# B&R Automation Studio project NAELD004C00R10L518F00 (part 7)

#### Act_OptP0001Startup.st
```iecst
ACTION Act_OptP0001Startup:

	//Screen Saver
	p_tyP0000SSaver ACCESS ADR(tyP0000SSaver.tySSaver);

	IF (eChgPage = UIP0001Startup) AND (eCurrPage = UIP0001Startup) THEN

		eStartupAct		:= StartupActRun;

		IF p_eStartupStat = StartupActRun AND p_eStartupStatus = Done THEN
			eStartupAct	:= StartupActIdle;

			IF p_bAlarmErr OR p_bAlarmWarning THEN
				eChgPage	:= UIP0600Alm;
			ELSE
				eChgPage	:= UIP0002Menu;
			END_IF

		END_IF

	END_IF

	tyP0001Startup.tyStartup.tyBarGraphStartup.iValue	:= DINT_TO_INT(p_eStartupStep + 1);
	tyP0001Startup.tyStartup.tyTxtStartupStat.sTxt		:= p_sStartupStepTxt;

	//IP Config
	IF DiagCpuIsSimulated() = FALSE THEN
		IF p_eStartupStep>1 THEN

			IF p_bStartupGetConfigDone THEN
				IF bTempAddrFillDone=FALSE THEN

					tyMcParamWr:= p_tyMcParamCurr;

					sTempIPAddr 	:= p_sHWInfoIPAddr;
					sTempSubnetMask	:= p_sHWInfoSubnetMask;
					udiTempEthMode	:= p_udiHWInfoEthMode;

					bTempAddrFillDone	:= TRUE;
				END_IF
			END_IF

			IF bTempAddrFillDone THEN

				IF bIPConfigChgDone=FALSE THEN

					IF  (p_tyMcParamCurr.eNetworkMod = UDINT_TO_DINT(udiTempEthMode)) AND (p_tyMcParamCurr.sIPAddr = sTempIPAddr) AND (p_tyMcParamCurr.sSubnetMask = sTempSubnetMask) THEN

						p_tyC0008MsgBox ACCESS ADR(tyP0001Startup.tyMsgBoxHide);
					ELSE
						IF p_bStartupMismatchSetConfigDone THEN

							IF (p_tyMcParamCurr.eNetworkMod <> UDINT_TO_DINT(udiTempEthMode)) THEN
								tyP0001Startup.tyMsgBoxIPConfig.tyTxtMsg.usiValueIdx := 114;
							ELSIF (p_tyMcParamCurr.sIPAddr <> sTempIPAddr) AND (p_tyMcParamCurr.sSubnetMask <> sTempSubnetMask) THEN
								tyP0001Startup.tyMsgBoxIPConfig.tyTxtMsg.usiValueIdx := 113;
							ELSIF (p_tyMcParamCurr.sIPAddr <> sTempIPAddr) THEN
								tyP0001Startup.tyMsgBoxIPConfig.tyTxtMsg.usiValueIdx := 111;
							ELSE
								tyP0001Startup.tyMsgBoxIPConfig.tyTxtMsg.usiValueIdx := 112;
							END_IF

							p_tyC0008MsgBox ACCESS ADR(tyP0001Startup.tyMsgBoxIPConfig);

						ELSE
							sSetIPAddr				:= p_tyMcParamCurr.sIPAddr;
							sSetSubnetMask			:= p_tyMcParamCurr.sSubnetMask;
							usiNetworkModeSelected	:= DINT_TO_USINT(p_tyMcParamCurr.eNetworkMod);

							bMismatchOverWriteConfig			:= TRUE;
						END_IF

					END_IF
				END_IF
			END_IF
		END_IF
	END_IF

	IF tyP0001Startup.tyMsgBoxIPConfig.tyBtnYes.bRtCompl = TRUE THEN
		tyP0001Startup.tyMsgBoxIPConfig.tyBtnYes.bRtCompl	:= FALSE;
		tyP0001Startup.tyMsgBoxIPConfig.tyBtnYes.bValue	:= FALSE;

		bIPConfigChgDone	:= TRUE;

		p_tyC0008MsgBox ACCESS ADR(tyP0001Startup.tyMsgBoxHide);

	ELSIF tyP0001Startup.tyMsgBoxIPConfig.tyBtnNo.bRtCompl = TRUE THEN

		IF (p_tyMcParamCurr.eNetworkMod <> UDINT_TO_DINT(udiTempEthMode))  THEN

			IF udiTempEthMode = DINT_TO_UDINT(IPFromDHCPServer) THEN

				bOverwriteEthMode	:= TRUE;
				bOverwriteIP 		:= FALSE;
				bOverwriteSubnet	:= FALSE;

				usiNetworkModeSelected	:= UDINT_TO_USINT(udiTempEthMode);

				tyMcParamWr.eNetworkMod	:= UDINT_TO_DINT(udiTempEthMode);

				bIPConfigChgDone	:= TRUE;

				tyP0001Startup.tyMsgBoxIPConfig.tyBtnNo.bRtCompl:= FALSE;
				tyP0001Startup.tyMsgBoxIPConfig.tyBtnNo.bValue	:= FALSE;

				p_tyC0008MsgBox ACCESS ADR(tyP0001Startup.tyMsgBoxHide);
			ELSE
				bOverwriteEthMode	:= TRUE;
				bOverwriteIP 		:= TRUE;
				bOverwriteSubnet	:= TRUE;

				usiNetworkModeSelected	:= UDINT_TO_USINT(udiTempEthMode);
				sSetIPAddr				:= sTempIPAddr;
				sSetSubnetMask			:= sTempSubnetMask;

				tyMcParamWr.eNetworkMod			:= UDINT_TO_DINT(udiTempEthMode);
				tyMcParamWr.sIPAddr				:= sTempIPAddr;
				tyMcParamWr.sSubnetMask			:= sTempSubnetMask;

				bIPConfigChgDone	:= TRUE;

				tyP0001Startup.tyMsgBoxIPConfig.tyBtnNo.bRtCompl:= FALSE;
				tyP0001Startup.tyMsgBoxIPConfig.tyBtnNo.bValue	:= FALSE;

				p_tyC0008MsgBox ACCESS ADR(tyP0001Startup.tyMsgBoxHide);
			END_IF

		ELSE

			IF (p_tyMcParamCurr.sIPAddr <> sTempIPAddr) AND (p_tyMcParamCurr.sSubnetMask <> sTempSubnetMask) THEN

				bOverwriteEthMode	:= FALSE;
				bOverwriteIP 		:= TRUE;
				bOverwriteSubnet	:= TRUE;

				sSetIPAddr		:= sTempIPAddr;
				sSetSubnetMask	:= sTempSubnetMask;

				tyMcParamWr.sIPAddr				:= sTempIPAddr;
				tyMcParamWr.sSubnetMask			:= sTempSubnetMask;

				bIPConfigChgDone	:= TRUE;

				tyP0001Startup.tyMsgBoxIPConfig.tyBtnNo.bRtCompl	:= FALSE;
				tyP0001Startup.tyMsgBoxIPConfig.tyBtnNo.bValue	:= FALSE;

				p_tyC0008MsgBox ACCESS ADR(tyP0001Startup.tyMsgBoxHide);

			ELSIF (p_tyMcParamCurr.sIPAddr <> sTempIPAddr) THEN

				bOverwriteEthMode	:= FALSE;
				bOverwriteIP 		:= TRUE;
				bOverwriteSubnet	:= FALSE;

				sSetIPAddr			:= sTempIPAddr;

				tyMcParamWr.sIPAddr	:= sTempIPAddr;

				bIPConfigChgDone	:= TRUE;

				tyP0001Startup.tyMsgBoxIPConfig.tyBtnNo.bRtCompl	:= FALSE;
				tyP0001Startup.tyMsgBoxIPConfig.tyBtnNo.bValue	:= FALSE;

				p_tyC0008MsgBox ACCESS ADR(tyP0001Startup.tyMsgBoxHide);
			ELSE

				bOverwriteEthMode	:= FALSE;
				bOverwriteIP 		:= FALSE;
				bOverwriteSubnet	:= TRUE;

				sSetSubnetMask	:= sTempSubnetMask;

				tyMcParamWr.sSubnetMask			:= sTempSubnetMask;

				bIPConfigChgDone				:= TRUE;

				tyP0001Startup.tyMsgBoxIPConfig.tyBtnNo.bRtCompl	:= FALSE;
				tyP0001Startup.tyMsgBoxIPConfig.tyBtnNo.bValue		:= FALSE;

				p_tyC0008MsgBox ACCESS ADR(tyP0001Startup.tyMsgBoxHide);
			END_IF
		END_IF
	END_IF

	//new for Hermes 1.3
	IF p_eStartupStep = StartupStepHermes AND p_bWaitDecision AND p_tyNtParamCurr.bHermesSvyPrep AND p_tyMcParamCurr.bHermesSvyEn AND p_tyNtParamCurr.bHermesSvyFirstMcInTheLine AND p_tyHermesConfiguration.tySvyParam.bFeatureQueryWorkOrderInfo THEN
		p_tyC0008MsgBox ACCESS ADR(tyP0001Startup.tyMsgBoxWorkOrder);

		IF tyP0001Startup.tyMsgBoxWorkOrder.tyBtnYes.bRtCompl = TRUE THEN
			tyP0001Startup.tyMsgBoxWorkOrder.tyBtnYes.bRtCompl	:= FALSE;
			bReadWorkOrder :=TRUE;
		END_IF

		IF tyP0001Startup.tyMsgBoxWorkOrder.tyBtnNo.bRtCompl = TRUE THEN
			tyP0001Startup.tyMsgBoxWorkOrder.tyBtnNo.bRtCompl	:= FALSE;
			bSkipWorkOrder :=TRUE;
		END_IF

		IF bReadWorkOrder OR bSkipWorkOrder THEN
			p_tyC0008MsgBox ACCESS ADR(tyP0001Startup.tyMsgBoxHide);
		END_IF

	ELSIF p_eStartupStep = StartupStepHermes AND p_bWaitDecision AND (p_tyNtParamCurr.bHermesSvyPrep = FALSE OR p_tyMcParamCurr.bHermesSvyEn = FALSE OR p_tyNtParamCurr.bHermesSvyFirstMcInTheLine = FALSE OR p_tyHermesConfiguration.tySvyParam.bFeatureQueryWorkOrderInfo = FALSE) THEN
		p_tyC0008MsgBox ACCESS ADR(tyP0001Startup.tyMsgBoxHide);
		bReadWorkOrder :=FALSE;
		bSkipWorkOrder :=TRUE;
	END_IF

END_ACTION
```

#### Act_EntP0002Disp.st
```iecst
ACTION Act_EntP0002Disp:

	//Access
	p_tyC0005Main ACCESS ADR(tyCommon.tyMain);

	p_tyC0007Notif ACCESS ADR(tyCommon.tyNotif);

	IF NOT bPromptSessionExp THEN
		p_tyC0008MsgBox ACCESS ADR(tyP0002Menu.tyMsgBoxHide);
	END_IF

	p_tyC0009Info ACCESS ADR(tyCommon.tyInfo);

	p_tyP0002Menu ACCESS ADR(tyP0002Menu.tyMenu);

	//Display
	//Leader Follower
	IF p_tyNtParamCurr.bLFPrep = TRUE AND p_tyMcParamCurr.bLFEn = TRUE AND ((NOT p_tyNtParamCurr.bLFUsrSetPrep AND p_tyNtParamCurr.bLeaderMc) OR (p_tyNtParamCurr.bLFUsrSetPrep AND p_tyMcParamCurr.bLFLeaderMc)) THEN
		fUIInRtStatOff(ADR(tyP0002Menu.tyMenu.tyBtnLFSet.uiRtStat));
		fUIInRtStatOff(ADR(tyP0002Menu.tyMenu.tyBtnLFCtrl.uiRtStat));
	ELSE
		fUIInRtStatHide(ADR(tyP0002Menu.tyMenu.tyBtnLFSet.uiRtStat));
		fUIInRtStatHide(ADR(tyP0002Menu.tyMenu.tyBtnLFCtrl.uiRtStat));
	END_IF

//	tyP0002Menu.tyMenu.tyBtnSimu.uiRtStat.0 := NOT(p_tyNtParamCurr.bProjAGVPrep AND p_tyMcParamCurr.bAGVComEn);

	//Login Logout Display
	IF bLoginSuccess = FALSE THEN
		tyP0002Menu.tyMenu.tyBtnLogin.usiBitmapIdx	:= 0;
		tyP0002Menu.tyMenu.tyBtnLogin.usiTxtIdx		:= 0;
	ELSE
		tyP0002Menu.tyMenu.tyBtnLogin.usiBitmapIdx	:= 1;
		tyP0002Menu.tyMenu.tyBtnLogin.usiTxtIdx		:= 1;
	END_IF

	//Mask
	Act_OptP0002Mask;
	bTeachServo := FALSE;
END_ACTION
```

#### Act_OptP0002ChgPage.st
```iecst
ACTION Act_OptP0002ChgPage:

	//General
	IF tyP0002Menu.tyMenu.tyBtnOpt.bRtCompl = TRUE THEN
		tyP0002Menu.tyMenu.tyBtnOpt.bRtCompl				:= FALSE;
		eChgPage											:= UIP0200OpsGen;

	ELSIF tyP0002Menu.tyMenu.tyBtnProdSel.bRtCompl = TRUE THEN
		tyP0002Menu.tyMenu.tyBtnProdSel.bRtCompl			:= FALSE;
		eChgPage											:= UIP0400ProdSel;

	ELSIF tyP0002Menu.tyMenu.tyBtnMagSel.bRtCompl = TRUE THEN
		tyP0002Menu.tyMenu.tyBtnMagSel.bRtCompl				:= FALSE;
		eChgPage											:= UIP0410MagSel;

	ELSIF tyP0002Menu.tyMenu.tyBtnMcInfo.bRtCompl = TRUE THEN
		tyP0002Menu.tyMenu.tyBtnMcInfo.bRtCompl				:= FALSE;
		eChgPage											:= UIP0300McInfo;

	ELSIF tyP0002Menu.tyMenu.tyBtnAlm.bRtCompl = TRUE THEN
		tyP0002Menu.tyMenu.tyBtnAlm.bRtCompl				:= FALSE;
		eChgPage											:= UIP0600Alm;

	ELSIF tyP0002Menu.tyMenu.tyBtnLogin.bRtCompl = TRUE THEN
		tyP0002Menu.tyMenu.tyBtnLogin.bRtCompl				:= FALSE;
		eChgPage											:= UIP0100Login;

	ELSIF tyP0002Menu.tyMenu.tyBtnLFCtrl.bRtCompl = TRUE THEN
		tyP0002Menu.tyMenu.tyBtnLFCtrl.bRtCompl				:= FALSE;
		eChgPage											:= UIP0700LFCtrl;

	ELSIF tyP0002Menu.tyMenu.tyBtnMagInfo.bRtCompl = TRUE THEN
		tyP0002Menu.tyMenu.tyBtnMagInfo.bRtCompl			:= FALSE;
		eChgPage											:= UIP0800MagInfo;

	//Manual
	ELSIF tyP0002Menu.tyMenu.tyBtnGenInput.bRtCompl = TRUE THEN
		bUIManualMod										:= TRUE;
		tyP0002Menu.tyMenu.tyBtnGenInput.bRtCompl			:= FALSE;
		eChgPage											:= UIP0900GenIn;

	ELSIF tyP0002Menu.tyMenu.tyBtnGenOutput.bRtCompl = TRUE THEN
		bUIManualMod										:= TRUE;
		tyP0002Menu.tyMenu.tyBtnGenOutput.bRtCompl			:= FALSE;
		eChgPage											:= UIP0910GenOut;

	ELSIF tyP0002Menu.tyMenu.tyBtnMovCtrl.bRtCompl = TRUE THEN
		bUIManualMod										:= TRUE;
		tyP0002Menu.tyMenu.tyBtnMovCtrl.bRtCompl			:= FALSE;
		eChgPage											:= UIP0920MtrNPneuCtrl;

	ELSIF tyP0002Menu.tyMenu.tyBtnCommCtrl.bRtCompl = TRUE THEN
		bUIManualMod										:= TRUE;
		tyP0002Menu.tyMenu.tyBtnCommCtrl.bRtCompl			:= FALSE;
		eChgPage											:= UIP0940CommCtrl;

	ELSIF tyP0002Menu.tyMenu.tyBtnSimu.bRtCompl = TRUE THEN
		tyP0002Menu.tyMenu.tyBtnSimu.bRtCompl				:= FALSE;
		eChgPage											:= UIP0950Simu;

	//Settings
	ELSIF tyP0002Menu.tyMenu.tyBtnLang.bRtCompl = TRUE THEN
		tyP0002Menu.tyMenu.tyBtnLang.bRtCompl				:= FALSE;
		eChgPage											:= UIP1000Lang;

	ELSIF tyP0002Menu.tyMenu.tyBtnMcSet.bRtCompl = TRUE THEN
		tyP0002Menu.tyMenu.tyBtnMcSet.bRtCompl				:= FALSE;
		eChgPage											:= UIP1020McSetNavi;

	ELSIF tyP0002Menu.tyMenu.tyBtnMagSet.bRtCompl = TRUE THEN
		tyP0002Menu.tyMenu.tyBtnMagSet.bRtCompl				:= FALSE;
		eChgPage											:= UIP1030MagSet;

	ELSIF tyP0002Menu.tyMenu.tyBtnProdSet.bRtCompl = TRUE THEN
		tyP0002Menu.tyMenu.tyBtnProdSet.bRtCompl			:= FALSE;
		eChgPage											:= UIP1040ProdSet;

	ELSIF tyP0002Menu.tyMenu.tyBtnLFSet.bRtCompl = TRUE THEN
		tyP0002Menu.tyMenu.tyBtnLFSet.bRtCompl				:= FALSE;
		eChgPage											:= UIP1050LFSet;

	ELSIF tyP0002Menu.tyMenu.tyBtnUsrMgmt.bRtCompl = TRUE THEN
		tyP0002Menu.tyMenu.tyBtnUsrMgmt.bRtCompl			:= FALSE;
		eChgPage											:= UIP1080UsrMgmt;

	END_IF
	fbActSimuTmr (IN:= tyP0002Menu.tyMenu.tyBtnHotspotActSimu.bValue = TRUE ,PT:=T#8s);
	IF fbActSimuTmr.Q THEN
		IF tyP0002Menu.tyMenu.tyBtnSimu.uiRtStat =0 THEN
			tyP0002Menu.tyMenu.tyBtnSimu.uiRtStat := 1;
			fbActSimuTmr (IN:= FALSE);
		ELSE
			tyP0002Menu.tyMenu.tyBtnSimu.uiRtStat := 0;
			fbActSimuTmr (IN:= FALSE);
		END_IF
	END_IF

END_ACTION
```

#### Act_OptP0002Mask.st
```iecst
ACTION Act_OptP0002Mask:

	tyP0002Menu.tyMenu.tyBtnOpt.uiMaskRtStat.0 					:= p_tyUsrMgmtCurrAccessRgt.bOpt;
	tyP0002Menu.tyMenu.tyBtnMcInfo.uiMaskRtStat.0 				:= p_tyUsrMgmtCurrAccessRgt.bMcInfo;
	tyP0002Menu.tyMenu.tyBtnMagInfo.uiMaskRtStat.0				:= p_tyUsrMgmtCurrAccessRgt.bMagInfo;
	tyP0002Menu.tyMenu.tyBtnAlm.uiMaskRtStat.0 					:= p_tyUsrMgmtCurrAccessRgt.bAlm;
	tyP0002Menu.tyMenu.tyBtnLogin.uiMaskRtStat.0				:= p_bOpsStatusStop;
	tyP0002Menu.tyMenu.tyBtnLFCtrl.uiMaskRtStat.0 				:= p_tyUsrMgmtCurrAccessRgt.bLFCtrl;
	tyP0002Menu.tyMenu.tyBtnGenInput.uiMaskRtStat.0				:= p_tyUsrMgmtCurrAccessRgt.bManual AND p_bOpsStatusStop;
	tyP0002Menu.tyMenu.tyBtnGenOutput.uiMaskRtStat.0			:= p_tyUsrMgmtCurrAccessRgt.bManual AND p_bOpsStatusStop;
	tyP0002Menu.tyMenu.tyBtnMovCtrl.uiMaskRtStat.0 				:= p_tyUsrMgmtCurrAccessRgt.bManual AND p_bOpsStatusStop;
	tyP0002Menu.tyMenu.tyBtnCommCtrl.uiMaskRtStat.0 			:= p_tyUsrMgmtCurrAccessRgt.bManual AND p_bOpsStatusStop;
	tyP0002Menu.tyMenu.tyBtnSimu.uiMaskRtStat.0 				:= p_tyUsrMgmtCurrAccessRgt.bSimulation AND p_bOpsStatusStop;
	tyP0002Menu.tyMenu.tyBtnProdSet.uiMaskRtStat.0 				:= p_tyUsrMgmtCurrAccessRgt.bProdSet AND p_bOpsStatusStop;
	tyP0002Menu.tyMenu.tyBtnMagSet.uiMaskRtStat.0				:= p_tyUsrMgmtCurrAccessRgt.bMagSet AND p_bOpsStatusStop;
	tyP0002Menu.tyMenu.tyBtnMcSet.uiMaskRtStat.0 				:= p_tyUsrMgmtCurrAccessRgt.bMcSet AND p_bOpsStatusStop;
	tyP0002Menu.tyMenu.tyBtnLang.uiMaskRtStat.0 				:= p_tyUsrMgmtCurrAccessRgt.bLang AND p_bOpsStatusStop;
	tyP0002Menu.tyMenu.tyBtnUsrMgmt.uiMaskRtStat.0 				:= p_tyUsrMgmtCurrAccessRgt.bUsrMgmt AND p_bOpsStatusStop;
	tyP0002Menu.tyMenu.tyBtnLFSet.uiMaskRtStat.0 				:= p_tyUsrMgmtCurrAccessRgt.bLFSet AND p_bOpsStatusStop;

	tyP0002Menu.tyMenu.tyBitmapMaskProdSetLCS.uiMaskRtStat.0	:= NOT(p_tyNtParamCurr.bLCSManageRcpPrep AND p_tyMcParamCurr.bLCSManageRcpEn);

//	IF p_tyNtParamCurr.eProjMag = LDMagTriple THEN
//		tyP0002Menu.tyMenu.tyBtnProdSel.uiMaskRtStat.0 	:= p_tyUsrMgmtCurrAccessRgt.bProdSel AND p_bOpsStatusStop AND NOT(p_bBuffer1MagPresent OR p_bBuffer2MagPresent OR p_bBuffer3MagPresent);
//		tyP0002Menu.tyMenu.tyBtnMagSel.uiMaskRtStat.0	:= p_tyUsrMgmtCurrAccessRgt.bMagSel AND p_bOpsStatusStop AND NOT(p_bBuffer1MagPresent OR p_bBuffer2MagPresent OR p_bBuffer3MagPresent);
//	ELSE
//		tyP0002Menu.tyMenu.tyBtnProdSel.uiMaskRtStat.0 	:= p_tyUsrMgmtCurrAccessRgt.bProdSel AND p_bOpsStatusStop AND NOT(p_bBuffer1MagPresent OR p_bBuffer2MagPresent);
//		tyP0002Menu.tyMenu.tyBtnMagSel.uiMaskRtStat.0	:= p_tyUsrMgmtCurrAccessRgt.bMagSel AND p_bOpsStatusStop AND NOT(p_bBuffer1MagPresent OR p_bBuffer2MagPresent);
//	END_IF

	IF p_tyNtParamCurr.eProjMag = LDMagTriple THEN
		tyP0002Menu.tyMenu.tyBtnProdSel.uiMaskRtStat.0 	:= p_bOpsStatusStop AND NOT(p_bBuffer1MagPresent OR p_bBuffer2MagPresent OR p_bBuffer3MagPresent);
		tyP0002Menu.tyMenu.tyBtnMagSel.uiMaskRtStat.0	:= p_bOpsStatusStop AND NOT(p_bBuffer1MagPresent OR p_bBuffer2MagPresent OR p_bBuffer3MagPresent);
	ELSIF p_tyNtParamCurr.eProjMag = LDMagQuadruple THEN
		tyP0002Menu.tyMenu.tyBtnProdSel.uiMaskRtStat.0 	:= p_bOpsStatusStop AND NOT(p_bBuffer1MagPresent OR p_bBuffer2MagPresent OR p_bBuffer3MagPresent OR p_bBuffer4MagPresent);
		tyP0002Menu.tyMenu.tyBtnMagSel.uiMaskRtStat.0	:= p_bOpsStatusStop AND NOT(p_bBuffer1MagPresent OR p_bBuffer2MagPresent OR p_bBuffer3MagPresent OR p_bBuffer4MagPresent);

	ELSE
		tyP0002Menu.tyMenu.tyBtnProdSel.uiMaskRtStat.0 	:= p_bOpsStatusStop AND NOT(p_bBuffer1MagPresent OR p_bBuffer2MagPresent);
		tyP0002Menu.tyMenu.tyBtnMagSel.uiMaskRtStat.0	:= p_bOpsStatusStop AND NOT(p_bBuffer1MagPresent OR p_bBuffer2MagPresent);
	END_IF
END_ACTION
```

#### Act_OptP0002MsgGuide.st
```iecst
ACTION Act_OptP0002MsgGuide:

	//Display
	tyP0002Menu.tyMenu.tyHotspotProdSel.uiRtStat.0	:= tyP0002Menu.tyMenu.tyBtnProdSel.uiMaskRtStat.0;
	tyP0002Menu.tyMenu.tyHotspotMagSel.uiRtStat.0	:= tyP0002Menu.tyMenu.tyBtnMagSel.uiMaskRtStat.0;

	IF p_tyNtParamCurr.eProjMag = LDMagTriple THEN
		tyP0002Menu.tyMenu.tyHotspotProdSel.bRtLk	:= NOT(p_bBuffer1MagPresent OR p_bBuffer2MagPresent OR p_bBuffer3MagPresent);
		tyP0002Menu.tyMenu.tyHotspotMagSel.bRtLk	:= NOT(p_bBuffer1MagPresent OR p_bBuffer2MagPresent OR p_bBuffer3MagPresent);
	ELSE
		tyP0002Menu.tyMenu.tyHotspotProdSel.bRtLk	:= NOT(p_bBuffer1MagPresent OR p_bBuffer2MagPresent);
		tyP0002Menu.tyMenu.tyHotspotMagSel.bRtLk	:= NOT(p_bBuffer1MagPresent OR p_bBuffer2MagPresent);
	END_IF

	//Control
	IF tyP0002Menu.tyMenu.tyHotspotProdSel.bRtCompl OR tyP0002Menu.tyMenu.tyHotspotMagSel.bRtCompl THEN
		p_tyC0008MsgBox ACCESS ADR(tyP0002Menu.tyMsgBoxRemoveMag);

		IF tyP0002Menu.tyMsgBoxRemoveMag.tyBtnNo.bRtCompl = TRUE THEN
			tyP0002Menu.tyMsgBoxRemoveMag.tyBtnNo.bRtCompl	:= FALSE;
			tyP0002Menu.tyMsgBoxRemoveMag.tyBtnNo.bValue	:= FALSE;

			p_tyC0008MsgBox ACCESS ADR(tyP0002Menu.tyMsgBoxHide);

			IF tyP0002Menu.tyMenu.tyHotspotProdSel.bRtCompl AND tyP0002Menu.tyMenu.tyBtnProdSel.uiMaskRtStat.0 THEN
				eChgPage	:= UIP0400ProdSel;

			ELSIF tyP0002Menu.tyMenu.tyHotspotMagSel.bRtCompl AND tyP0002Menu.tyMenu.tyBtnMagSel.uiMaskRtStat.0 THEN
				eChgPage	:= UIP0410MagSel;

			END_IF

			tyP0002Menu.tyMenu.tyHotspotProdSel.bRtCompl	:= FALSE;
			tyP0002Menu.tyMenu.tyHotspotMagSel.bRtCompl		:= FALSE;

		END_IF

	END_IF

END_ACTION
```

#### Act_OptP0002ToP1081UnlockCoverPB.st
```iecst
ACTION Act_OptP0002ToP1081UnlockCoverPB:

	IF p_tyDI.bDSUnlockCoverSig AND (p_bOpsTravLifStandby OR p_bOpsRun = FALSE) AND p_ePullConvStatus <> Busy THEN
		bMachineSafetySigToDS := TRUE;																						//
	ELSE
		bMachineSafetySigToDS := FALSE;																						//
	END_IF

END_ACTION
```

#### Act_EntP0200Disp.st
```iecst
ACTION Act_EntP0200Disp:

	//Access Address
	p_tyC0005Main ACCESS ADR(tyCommon.tyMain);

	p_tyC0007Notif ACCESS ADR(tyCommon.tyNotif);

	p_tyC0008MsgBox ACCESS ADR(tyP0200OpsGen.tyMsgBoxHide);

	p_tyC0009Info ACCESS ADR(tyCommon.tyInfo);

	p_tyC0010RcyMsg ACCESS ADR(tyP0200OpsGen.tyRcyMsgHide);

	p_tyP0200OpsGen ACCESS ADR(tyP0200OpsGen.tyOps);
	p_tyP0200OpsDSCommB ACCESS ADR(tyP0200OpsGen.tyDSCommB);

	p_tyP0200OpsDSAVSMEMA ACCESS ADR(tyP0200OpsGen.tyDSAVSMEMA);
	p_tyP0200OpsDSBVSMEMA ACCESS ADR(tyP0200OpsGen.tyDSBVSMEMA);
	p_tyP0200OpsDSAVSMEMA1 ACCESS ADR(tyP0200OpsGen.tyDSAVSMEMA1);
	p_tyP0200OpsDSBVSMEMA1 ACCESS ADR(tyP0200OpsGen.tyDSBVSMEMA1);
	p_tyP0200OpsBypsInitConv ACCESS ADR(tyP0200OpsGen.tyBypsInitConv);

	p_tyP0200OpsBarCodeScan ACCESS ADR(tyP0200OpsGen.tyBarCodeScan);
	//Display
	//Downstream A
	IF p_tyMcParamCurr.eDSCommA = McSetCommModHermes THEN
		tyP0200OpsGen.tyOps.tyBitmapDSAComm.usiValueIdx	:= 1;
		tyP0200OpsGen.tyOps.tyBitmapDSAComm1.usiValueIdx	:= 1;
	ELSIF p_tyMcParamCurr.eDSCommA = McSetCommModSMEMA THEN
		tyP0200OpsGen.tyOps.tyBitmapDSAComm.usiValueIdx	:= 0;
		tyP0200OpsGen.tyOps.tyBitmapDSAComm1.usiValueIdx	:= 0;
	END_IF

	//Downstream B
	IF p_tyMcParamCurr.eDSCommB = McSetCommModHermes THEN
		tyP0200OpsGen.tyDSCommB.tyBitmapDSBComm.usiValueIdx	:= 1;
		tyP0200OpsGen.tyDSCommB.tyBitmapDSBComm1.usiValueIdx	:= 1;
	ELSIF p_tyMcParamCurr.eDSCommB = McSetCommModSMEMA THEN
		tyP0200OpsGen.tyDSCommB.tyBitmapDSBComm.usiValueIdx	:= 0;
		tyP0200OpsGen.tyDSCommB.tyBitmapDSBComm1.usiValueIdx	:= 0;
	END_IF

	//Virtual SMEMA
	IF (p_tyUsrMgmtCurrUsr.eUsrLvl = UsrMgmtLvl1) OR p_tyNtParamCurr.bVSMEMAPrep = FALSE OR p_tyMcParamCurr.bVSMEMAEn = FALSE OR (p_tyMcParamCurr.eDSCommA = McSetCommModHermes AND p_tyMcParamCurr.eDSCommB = McSetCommModHermes) THEN

		tyP0200OpsGen.tyOps.tyHotspotDSAVSMEMA.bValue		:= FALSE;
		tyP0200OpsGen.tyDSCommB.tyHotspotDSBVSMEMA.bValue	:= FALSE;
		tyP0200OpsGen.tyOps.tyHotspotDSAVSMEMA1.bValue		:= FALSE;
		tyP0200OpsGen.tyDSCommB.tyHotspotDSBVSMEMA1.bValue	:= FALSE;

		memset(ADR(tyP0200OpsGen.tyDSAVSMEMA), 0, SIZEOF(tyP0200OpsGen.tyDSAVSMEMA));
		memset(ADR(tyP0200OpsGen.tyDSBVSMEMA), 0, SIZEOF(tyP0200OpsGen.tyDSBVSMEMA));
		memset(ADR(tyP0200OpsGen.tyDSAVSMEMA1), 0, SIZEOF(tyP0200OpsGen.tyDSAVSMEMA1));
		memset(ADR(tyP0200OpsGen.tyDSBVSMEMA1), 0, SIZEOF(tyP0200OpsGen.tyDSBVSMEMA1));

		fUIInRtStatHide(ADR(tyP0200OpsGen.tyOps.tyHotspotDSAVSMEMA.uiRtStat));
		fUIInRtStatHide(ADR(tyP0200OpsGen.tyDSCommB.tyHotspotDSBVSMEMA.uiRtStat));
		fUIInRtStatHide(ADR(tyP0200OpsGen.tyDSAVSMEMA.tyLyr.uiRtStat));
		fUIInRtStatHide(ADR(tyP0200OpsGen.tyDSBVSMEMA.tyLyr.uiRtStat));

		fUIInRtStatHide(ADR(tyP0200OpsGen.tyOps.tyHotspotDSAVSMEMA1.uiRtStat));
		fUIInRtStatHide(ADR(tyP0200OpsGen.tyDSCommB.tyHotspotDSBVSMEMA1.uiRtStat));
		fUIInRtStatHide(ADR(tyP0200OpsGen.tyDSAVSMEMA1.tyLyr.uiRtStat));
		fUIInRtStatHide(ADR(tyP0200OpsGen.tyDSBVSMEMA1.tyLyr.uiRtStat));

		bVSMEMADSAEn	:= FALSE;
		bVSMEMADSBEn	:= FALSE;
	ELSE

		//Downstream A
		IF p_tyMcParamCurr.eDSCommA = McSetCommModHermes THEN
			tyP0200OpsGen.tyOps.tyHotspotDSAVSMEMA.bValue	:= FALSE;
			tyP0200OpsGen.tyOps.tyHotspotDSAVSMEMA1.bValue	:= FALSE;

			memset(ADR(tyP0200OpsGen.tyDSAVSMEMA), 0, SIZEOF(tyP0200OpsGen.tyDSAVSMEMA));

			fUIInRtStatHide(ADR(tyP0200OpsGen.tyOps.tyHotspotDSAVSMEMA.uiRtStat));
			fUIInRtStatHide(ADR(tyP0200OpsGen.tyDSAVSMEMA.tyLyr.uiRtStat));

			memset(ADR(tyP0200OpsGen.tyDSAVSMEMA1), 0, SIZEOF(tyP0200OpsGen.tyDSAVSMEMA1));

			fUIInRtStatHide(ADR(tyP0200OpsGen.tyOps.tyHotspotDSAVSMEMA1.uiRtStat));
			fUIInRtStatHide(ADR(tyP0200OpsGen.tyDSAVSMEMA1.tyLyr.uiRtStat));

		ELSIF p_tyMcParamCurr.eDSCommA = McSetCommModSMEMA THEN
			IF p_tyNtParamCurr.bUIConvDirRL = FALSE THEN //LR
				fUIInRtStatOff(ADR(tyP0200OpsGen.tyOps.tyHotspotDSAVSMEMA.uiRtStat));

				fUIInRtStatHide(ADR(tyP0200OpsGen.tyOps.tyHotspotDSAVSMEMA1.uiRtStat));
				fUIInRtStatHide(ADR(tyP0200OpsGen.tyOps.tyTxtLane1.uiRtStat));
				fUIInRtStatHide(ADR(tyP0200OpsGen.tyOps.tyBitmapDSIn1.uiRtStat));
				fUIInRtStatHide(ADR(tyP0200OpsGen.tyOps.tyBitmapDSOut1.uiRtStat));
				fUIInRtStatHide(ADR(tyP0200OpsGen.tyOps.tyBitmapDSAComm1.uiRtStat));
				memset(ADR(tyP0200OpsGen.tyDSAVSMEMA1), 0, SIZEOF(tyP0200OpsGen.tyDSAVSMEMA1));
				fUIInRtStatHide(ADR(tyP0200OpsGen.tyDSAVSMEMA1.tyLyr.uiRtStat));
			ELSE //RL
				fUIInRtStatOff(ADR(tyP0200OpsGen.tyOps.tyHotspotDSAVSMEMA1.uiRtStat));

				fUIInRtStatHide(ADR(tyP0200OpsGen.tyOps.tyHotspotDSAVSMEMA.uiRtStat));
				fUIInRtStatHide(ADR(tyP0200OpsGen.tyOps.tyTxtLane.uiRtStat));
				fUIInRtStatHide(ADR(tyP0200OpsGen.tyOps.tyBitmapDSIn.uiRtStat));
				fUIInRtStatHide(ADR(tyP0200OpsGen.tyOps.tyBitmapDSOut.uiRtStat));
				fUIInRtStatHide(ADR(tyP0200OpsGen.tyOps.tyBitmapDSAComm.uiRtStat));
				memset(ADR(tyP0200OpsGen.tyDSAVSMEMA), 0, SIZEOF(tyP0200OpsGen.tyDSAVSMEMA));
				fUIInRtStatHide(ADR(tyP0200OpsGen.tyDSAVSMEMA.tyLyr.uiRtStat));

			END_IF

		END_IF

		//Downstream B
		IF p_tyNtParamCurr.bProjLaneBPrep THEN
			IF p_tyMcParamCurr.eDSCommB = McSetCommModHermes THEN
				tyP0200OpsGen.tyDSCommB.tyHotspotDSBVSMEMA.bValue	:= FALSE;
				tyP0200OpsGen.tyDSCommB.tyHotspotDSBVSMEMA1.bValue	:= FALSE;

				memset(ADR(tyP0200OpsGen.tyDSBVSMEMA), 0, SIZEOF(tyP0200OpsGen.tyDSBVSMEMA));
				fUIInRtStatHide(ADR(tyP0200OpsGen.tyDSCommB.tyHotspotDSBVSMEMA.uiRtStat));
				fUIInRtStatHide(ADR(tyP0200OpsGen.tyDSBVSMEMA.tyLyr.uiRtStat));

				memset(ADR(tyP0200OpsGen.tyDSBVSMEMA1), 0, SIZEOF(tyP0200OpsGen.tyDSBVSMEMA1));
				fUIInRtStatHide(ADR(tyP0200OpsGen.tyDSCommB.tyHotspotDSBVSMEMA1.uiRtStat));
				fUIInRtStatHide(ADR(tyP0200OpsGen.tyDSBVSMEMA1.tyLyr.uiRtStat));

			ELSIF p_tyMcParamCurr.eDSCommB = McSetCommModSMEMA THEN
				IF p_tyNtParamCurr.bUIConvDirRL = FALSE THEN //LR
					fUIInRtStatOff(ADR(tyP0200OpsGen.tyDSCommB.tyHotspotDSBVSMEMA.uiRtStat));

					fUIInRtStatHide(ADR(tyP0200OpsGen.tyDSCommB.tyHotspotDSBVSMEMA1.uiRtStat));
					fUIInRtStatHide(ADR(tyP0200OpsGen.tyDSCommB.tyTxtLane1.uiRtStat));
					fUIInRtStatHide(ADR(tyP0200OpsGen.tyDSCommB.tyBitmapIn1.uiRtStat));
					fUIInRtStatHide(ADR(tyP0200OpsGen.tyDSCommB.tyBitmapOut1.uiRtStat));
					fUIInRtStatHide(ADR(tyP0200OpsGen.tyDSCommB.tyBitmapDSBComm1.uiRtStat));
					fUIInRtStatHide(ADR(tyP0200OpsGen.tyDSBVSMEMA1.tyLyr.uiRtStat));

				ELSE
					fUIInRtStatOff(ADR(tyP0200OpsGen.tyDSCommB.tyHotspotDSBVSMEMA1.uiRtStat));

					fUIInRtStatHide(ADR(tyP0200OpsGen.tyDSCommB.tyHotspotDSBVSMEMA.uiRtStat));
					fUIInRtStatHide(ADR(tyP0200OpsGen.tyDSCommB.tyTxtLane.uiRtStat));
					fUIInRtStatHide(ADR(tyP0200OpsGen.tyDSCommB.tyBitmapIn.uiRtStat));
					fUIInRtStatHide(ADR(tyP0200OpsGen.tyDSCommB.tyBitmapOut.uiRtStat));
					fUIInRtStatHide(ADR(tyP0200OpsGen.tyDSCommB.tyBitmapDSBComm.uiRtStat));
					fUIInRtStatHide(ADR(tyP0200OpsGen.tyDSBVSMEMA.tyLyr.uiRtStat));
				END_IF

			END_IF

		END_IF

	END_IF

	//Conveyor Direction - SMEMA Arrow Indicator
	IF p_tyNtParamCurr.bUIConvDirRL THEN
		fUIInRtStatHide(ADR(tyP0200OpsGen.tyOps.tyBitmapDSIn.uiRtStat));
		fUIInRtStatHide(ADR(tyP0200OpsGen.tyOps.tyBitmapDSOut.uiRtStat));
		fUIInRtStatHide(ADR(tyP0200OpsGen.tyOps.tyTxtLane.uiRtStat));
		fUIInRtStatHide(ADR(tyP0200OpsGen.tyOps.tyHotspotDSAVSMEMA.uiRtStat));
		fUIInRtStatHide(ADR(tyP0200OpsGen.tyOps.tyBitmapDSAComm.uiRtStat));
		fUIInRtStatHide(ADR(tyP0200OpsGen.tyOps.tyBitmapDSAComm.uiMaskRtStat));

		fUIInRtStatHide(ADR(tyP0200OpsGen.tyDSCommB.tyBitmapIn.uiRtStat));
		fUIInRtStatHide(ADR(tyP0200OpsGen.tyDSCommB.tyBitmapOut.uiRtStat));
		fUIInRtStatHide(ADR(tyP0200OpsGen.tyDSCommB.tyTxtLane.uiRtStat));
		fUIInRtStatHide(ADR(tyP0200OpsGen.tyDSCommB.tyHotspotDSBVSMEMA.uiRtStat));
		fUIInRtStatHide(ADR(tyP0200OpsGen.tyDSCommB.tyBitmapDSBComm.uiRtStat));
		fUIInRtStatHide(ADR(tyP0200OpsGen.tyDSCommB.tyBitmapDSBComm.uiMaskRtStat));

		fUIInRtStatOff(ADR(tyP0200OpsGen.tyOps.tyBitmapDSIn1.uiRtStat));
		fUIInRtStatOff(ADR(tyP0200OpsGen.tyOps.tyBitmapDSOut1.uiRtStat));
		fUIInRtStatOff(ADR(tyP0200OpsGen.tyOps.tyTxtLane1.uiRtStat));
		fUIInRtStatOff(ADR(tyP0200OpsGen.tyOps.tyHotspotDSAVSMEMA1.uiRtStat));
		fUIInRtStatOff(ADR(tyP0200OpsGen.tyOps.tyBitmapDSAComm1.uiRtStat));
		fUIInRtStatOff(ADR(tyP0200OpsGen.tyOps.tyBitmapDSAComm1.uiMaskRtStat));

		fUIInRtStatOff(ADR(tyP0200OpsGen.tyDSCommB.tyBitmapIn1.uiRtStat));
		fUIInRtStatOff(ADR(tyP0200OpsGen.tyDSCommB.tyBitmapOut1.uiRtStat));
		fUIInRtStatOff(ADR(tyP0200OpsGen.tyDSCommB.tyTxtLane1.uiRtStat));
		fUIInRtStatOff(ADR(tyP0200OpsGen.tyDSCommB.tyHotspotDSBVSMEMA1.uiRtStat));
		fUIInRtStatOff(ADR(tyP0200OpsGen.tyDSCommB.tyBitmapDSBComm1.uiRtStat));
		fUIInRtStatOff(ADR(tyP0200OpsGen.tyDSCommB.tyBitmapDSBComm1.uiMaskRtStat));

	ELSE // LR

		fUIInRtStatOff(ADR(tyP0200OpsGen.tyOps.tyBitmapDSIn.uiRtStat));
		fUIInRtStatOff(ADR(tyP0200OpsGen.tyOps.tyBitmapDSOut.uiRtStat));
		fUIInRtStatOff(ADR(tyP0200OpsGen.tyOps.tyTxtLane.uiRtStat));
		fUIInRtStatOff(ADR(tyP0200OpsGen.tyOps.tyHotspotDSAVSMEMA.uiRtStat));
		fUIInRtStatOff(ADR(tyP0200OpsGen.tyOps.tyBitmapDSAComm.uiRtStat));
		fUIInRtStatOff(ADR(tyP0200OpsGen.tyOps.tyBitmapDSAComm.uiMaskRtStat));

		fUIInRtStatOff(ADR(tyP0200OpsGen.tyDSCommB.tyBitmapIn.uiRtStat));
		fUIInRtStatOff(ADR(tyP0200OpsGen.tyDSCommB.tyBitmapOut.uiRtStat));
		fUIInRtStatOff(ADR(tyP0200OpsGen.tyDSCommB.tyTxtLane.uiRtStat));
		fUIInRtStatOff(ADR(tyP0200OpsGen.tyDSCommB.tyHotspotDSBVSMEMA.uiRtStat));
		fUIInRtStatOff(ADR(tyP0200OpsGen.tyDSCommB.tyBitmapDSBComm.uiRtStat));
		fUIInRtStatOff(ADR(tyP0200OpsGen.tyDSCommB.tyBitmapDSBComm.uiMaskRtStat));

		fUIInRtStatHide(ADR(tyP0200OpsGen.tyOps.tyBitmapDSIn1.uiRtStat));
		fUIInRtStatHide(ADR(tyP0200OpsGen.tyOps.tyBitmapDSOut1.uiRtStat));
		fUIInRtStatHide(ADR(tyP0200OpsGen.tyOps.tyTxtLane1.uiRtStat));
		fUIInRtStatHide(ADR(tyP0200OpsGen.tyOps.tyHotspotDSAVSMEMA1.uiRtStat));
		fUIInRtStatHide(ADR(tyP0200OpsGen.tyOps.tyBitmapDSAComm1.uiRtStat));
		fUIInRtStatHide(ADR(tyP0200OpsGen.tyOps.tyBitmapDSAComm1.uiMaskRtStat));

		fUIInRtStatHide(ADR(tyP0200OpsGen.tyDSCommB.tyBitmapIn1.uiRtStat));
		fUIInRtStatHide(ADR(tyP0200OpsGen.tyDSCommB.tyBitmapOut1.uiRtStat));
		fUIInRtStatHide(ADR(tyP0200OpsGen.tyDSCommB.tyTxtLane1.uiRtStat));
		fUIInRtStatHide(ADR(tyP0200OpsGen.tyDSCommB.tyHotspotDSBVSMEMA1.uiRtStat));
		fUIInRtStatHide(ADR(tyP0200OpsGen.tyDSCommB.tyBitmapDSBComm1.uiRtStat));
		fUIInRtStatHide(ADR(tyP0200OpsGen.tyDSCommB.tyBitmapDSBComm1.uiMaskRtStat));

	END_IF

	//Disable AIV function
	IF p_tyMcParamCurr.bAGVComEn = FALSE THEN
		//	fUIInRtStatHide(ADR(tyP0200OpsGen.tyOps.tyHotspotOpsAIV.uiRtStat));
		fUIInRtStatOff(ADR(tyP0200OpsGen.tyOps.tyHotspotOpsAIV.uiMaskRtStat));
	ELSE
		fUIInRtStatHide(ADR(tyP0200OpsGen.tyOps.tyHotspotOpsAIV.uiMaskRtStat));
	END_IF

	//Barcode Scanner
	tyP0200OpsGen.tyOps.tyBtnBarCodeScan.uiRtStat.0 := NOT ((p_tyNtParamCurr.bUSBScannerPrep OR  p_tyNtParamCurr.bRS232ScannerPrep) AND p_tyMcParamCurr.bScannerEn);
	tyP0200OpsGen.tyOps.tyBitmapBarCodeScan.uiRtStat.0 := NOT ((p_tyNtParamCurr.bUSBScannerPrep OR  p_tyNtParamCurr.bRS232ScannerPrep) AND p_tyMcParamCurr.bScannerEn);

	tyP0200OpsGen.tyBarCodeScan.tyStringBarCode.sValue  := '';

END_ACTION
```

#### Act_OptP0200ChgPage.st
```iecst
ACTION Act_OptP0200ChgPage:

	IF tyP0200OpsGen.tyOps.tyHotspotOpsTravLifter.bRtCompl = TRUE THEN
		tyP0200OpsGen.tyOps.tyHotspotOpsTravLifter.bRtCompl	:= FALSE;

		eChgPage	:= UIP0201OpsTravLifter;

	ELSIF tyP0200OpsGen.tyOps.tyHotspotOps2Mag1.bRtCompl = TRUE OR tyP0200OpsGen.tyOps.tyHotspotOps3Mag1.bRtCompl = TRUE
		OR tyP0200OpsGen.tyOps.tyHotspotOps4Mag1.bRtCompl = TRUE
		THEN
		tyP0200OpsGen.tyOps.tyHotspotOps2Mag1.bRtCompl	:= FALSE;
		tyP0200OpsGen.tyOps.tyHotspotOps3Mag1.bRtCompl	:= FALSE;
		tyP0200OpsGen.tyOps.tyHotspotOps4Mag1.bRtCompl	:= FALSE;
		eChgPage	:= UIP0202OpsMag1;

	ELSIF tyP0200OpsGen.tyOps.tyHotspotOps2Mag2.bRtCompl = TRUE OR tyP0200OpsGen.tyOps.tyHotspotOps3Mag2.bRtCompl = TRUE
		OR tyP0200OpsGen.tyOps.tyHotspotOps4Mag2.bRtCompl = TRUE
		THEN
		tyP0200OpsGen.tyOps.tyHotspotOps2Mag2.bRtCompl	:= FALSE;
		tyP0200OpsGen.tyOps.tyHotspotOps3Mag2.bRtCompl	:= FALSE;
		tyP0200OpsGen.tyOps.tyHotspotOps4Mag2.bRtCompl	:= FALSE;
		eChgPage	:= UIP0203OpsMag2;

	ELSIF tyP0200OpsGen.tyOps.tyHotspotOps3Mag3.bRtCompl = TRUE OR tyP0200OpsGen.tyOps.tyHotspotOps4Mag3.bRtCompl = TRUE
		THEN
		tyP0200OpsGen.tyOps.tyHotspotOps3Mag3.bRtCompl	:= FALSE;
		tyP0200OpsGen.tyOps.tyHotspotOps4Mag3.bRtCompl	:= FALSE;
		eChgPage	:= UIP0204OpsMag3;

	ELSIF tyP0200OpsGen.tyOps.tyHotspotOps4Mag4.bRtCompl = TRUE
		THEN
		tyP0200OpsGen.tyOps.tyHotspotOps4Mag4.bRtCompl	:= FALSE;

		eChgPage	:= UIP0206OpsMag4;

	ELSIF tyP0200OpsGen.tyOps.tyHotspotOpsAIV.bRtCompl = TRUE THEN
		tyP0200OpsGen.tyOps.tyHotspotOpsAIV.bRtCompl	:= FALSE;

		eChgPage	:= UIP0205OpsAIV;

	ELSIF tyP0200OpsGen.tyOps.tyHotspotOpsMagInfo.bRtCompl = TRUE THEN
		tyP0200OpsGen.tyOps.tyHotspotOpsMagInfo.bRtCompl	:= FALSE;

		eChgPage	:= UIP0800MagInfo;

	END_IF

END_ACTION
```

#### Act_OptP0200UpdtDat.st
```iecst
ACTION Act_OptP0200UpdtDat:

	//PCB Status
	IF p_bPullConvHvBrd = TRUE THEN
		tyP0200OpsGen.tyOps.tyBitmapPCB.usiValueIdx	:= 1;
	ELSE
		tyP0200OpsGen.tyOps.tyBitmapPCB.usiValueIdx	:= 0;
	END_IF

	//Communication - Mask
	IF p_tyNtParamCurr.bUIConvDirRL = FALSE THEN
		fUIInRtStatHide(ADR(tyP0200OpsGen.tyOps.tyBitmapDSAComm1.uiMaskRtStat));
		fUIInRtStatHide(ADR(tyP0200OpsGen.tyDSCommB.tyBitmapDSBComm1.uiMaskRtStat));
		IF p_tyMcParamCurr.eDSCommA = McSetCommModSMEMA THEN
			fUIInRtStatHide(ADR(tyP0200OpsGen.tyOps.tyBitmapDSAComm.uiMaskRtStat));
		ELSIF p_tyMcParamCurr.eDSCommA = McSetCommModHermes THEN
			IF p_bDSHermesAConnected = TRUE THEN
				fUIInRtStatHide(ADR(tyP0200OpsGen.tyOps.tyBitmapDSAComm.uiMaskRtStat));
			ELSE
				fUIInRtStatOff(ADR(tyP0200OpsGen.tyOps.tyBitmapDSAComm.uiMaskRtStat));
			END_IF
		END_IF

		IF p_tyMcParamCurr.eDSCommB = McSetCommModSMEMA THEN
			fUIInRtStatHide(ADR(tyP0200OpsGen.tyDSCommB.tyBitmapDSBComm.uiMaskRtStat));
		ELSIF p_tyMcParamCurr.eDSCommB = McSetCommModHermes THEN
			IF p_bDSHermesBConnected = TRUE THEN
				fUIInRtStatHide(ADR(tyP0200OpsGen.tyDSCommB.tyBitmapDSBComm.uiMaskRtStat));
			ELSE
				fUIInRtStatOff(ADR(tyP0200OpsGen.tyDSCommB.tyBitmapDSBComm.uiMaskRtStat));
			END_IF
		END_IF
	ELSE
		fUIInRtStatHide(ADR(tyP0200OpsGen.tyOps.tyBitmapDSAComm.uiMaskRtStat));
		fUIInRtStatHide(ADR(tyP0200OpsGen.tyDSCommB.tyBitmapDSBComm.uiMaskRtStat));
		IF p_tyMcParamCurr.eDSCommA = McSetCommModSMEMA THEN
			fUIInRtStatHide(ADR(tyP0200OpsGen.tyOps.tyBitmapDSAComm1.uiMaskRtStat));
		ELSIF p_tyMcParamCurr.eDSCommA = McSetCommModHermes THEN
			IF p_bDSHermesAConnected = TRUE THEN
				fUIInRtStatHide(ADR(tyP0200OpsGen.tyOps.tyBitmapDSAComm1.uiMaskRtStat));
			ELSE
				fUIInRtStatOff(ADR(tyP0200OpsGen.tyOps.tyBitmapDSAComm1.uiMaskRtStat));
			END_IF
		END_IF

		IF p_tyMcParamCurr.eDSCommB = McSetCommModSMEMA THEN
			fUIInRtStatHide(ADR(tyP0200OpsGen.tyDSCommB.tyBitmapDSBComm1.uiMaskRtStat));
		ELSIF p_tyMcParamCurr.eDSCommB = McSetCommModHermes THEN
			IF p_bDSHermesBConnected = TRUE THEN
				fUIInRtStatHide(ADR(tyP0200OpsGen.tyDSCommB.tyBitmapDSBComm1.uiMaskRtStat));
			ELSE
				fUIInRtStatOff(ADR(tyP0200OpsGen.tyDSCommB.tyBitmapDSBComm1.uiMaskRtStat));
			END_IF
		END_IF
	END_IF
	//Communication - Signal
	//DBA A
	IF p_tyNtParamCurr.bUIConvDirRL = FALSE THEN
		IF p_tyMcParamCurr.eDSCommA = McSetCommModSMEMA THEN
			IF p_bDSSMEMAAUSRdy = TRUE THEN
				IF p_bDSSMEMAAUSGdBrdRdy = TRUE THEN
					tyP0200OpsGen.tyOps.tyBitmapDSOut.usiValueIdx	:= 1;
				ELSE
					tyP0200OpsGen.tyOps.tyBitmapDSOut.usiValueIdx	:= 2;
				END_IF
			ELSE
				tyP0200OpsGen.tyOps.tyBitmapDSOut.usiValueIdx	:= 0;
			END_IF

		ELSIF p_tyMcParamCurr.eDSCommA = McSetCommModHermes THEN
			IF p_bDSHermesAUSRdy = TRUE THEN
				IF p_bDSHermesAUSGdRdy = TRUE THEN
					tyP0200OpsGen.tyOps.tyBitmapDSOut.usiValueIdx	:= 1;
				ELSE
					tyP0200OpsGen.tyOps.tyBitmapDSOut.usiValueIdx	:= 2;
				END_IF
			ELSE
				tyP0200OpsGen.tyOps.tyBitmapDSOut.usiValueIdx	:= 0;
			END_IF

		END_IF
	ELSE
		IF p_tyMcParamCurr.eDSCommA = McSetCommModSMEMA THEN
			IF p_bDSSMEMAAUSRdy = TRUE THEN
				IF p_bDSSMEMAAUSGdBrdRdy = TRUE THEN
					tyP0200OpsGen.tyOps.tyBitmapDSOut1.usiValueIdx	:= 1;
				ELSE
					tyP0200OpsGen.tyOps.tyBitmapDSOut1.usiValueIdx	:= 2;
				END_IF
			ELSE
				tyP0200OpsGen.tyOps.tyBitmapDSOut1.usiValueIdx	:= 0;
			END_IF

		ELSIF p_tyMcParamCurr.eDSCommA = McSetCommModHermes THEN
			IF p_bDSHermesAUSRdy = TRUE THEN
				IF p_bDSHermesAUSGdRdy = TRUE THEN
					tyP0200OpsGen.tyOps.tyBitmapDSOut1.usiValueIdx	:= 1;
				ELSE
					tyP0200OpsGen.tyOps.tyBitmapDSOut1.usiValueIdx	:= 2;
				END_IF
			ELSE
				tyP0200OpsGen.tyOps.tyBitmapDSOut1.usiValueIdx	:= 0;
			END_IF

		END_IF
	END_IF

	//DSB A
	IF p_tyNtParamCurr.bUIConvDirRL = FALSE THEN
		IF p_tyMcParamCurr.eDSCommA = McSetCommModSMEMA THEN
			IF p_bDSSMEMAADSRdy = TRUE THEN
				tyP0200OpsGen.tyOps.tyBitmapDSIn.usiValueIdx	:= 1;
			ELSE
				tyP0200OpsGen.tyOps.tyBitmapDSIn.usiValueIdx	:= 0;
			END_IF

		ELSIF p_tyMcParamCurr.eDSCommA = McSetCommModHermes THEN
			IF p_bDSHermesADSRdy = TRUE THEN
				IF p_bDSHermesADSGdRdy = TRUE THEN
					tyP0200OpsGen.tyOps.tyBitmapDSIn.usiValueIdx	:= 1;
				ELSE
					tyP0200OpsGen.tyOps.tyBitmapDSIn.usiValueIdx	:= 2;
				END_IF
			ELSE
				tyP0200OpsGen.tyOps.tyBitmapDSIn.usiValueIdx	:= 0;
			END_IF

		END_IF
	ELSE
		IF p_tyMcParamCurr.eDSCommA = McSetCommModSMEMA THEN
			IF p_bDSSMEMAADSRdy = TRUE THEN
				tyP0200OpsGen.tyOps.tyBitmapDSIn1.usiValueIdx	:= 1;
			ELSE
				tyP0200OpsGen.tyOps.tyBitmapDSIn1.usiValueIdx	:= 0;
			END_IF

		ELSIF p_tyMcParamCurr.eDSCommA = McSetCommModHermes THEN
			IF p_bDSHermesADSRdy = TRUE THEN
				IF p_bDSHermesADSGdRdy = TRUE THEN
					tyP0200OpsGen.tyOps.tyBitmapDSIn1.usiValueIdx	:= 1;
				ELSE
					tyP0200OpsGen.tyOps.tyBitmapDSIn1.usiValueIdx	:= 2;
				END_IF
			ELSE
				tyP0200OpsGen.tyOps.tyBitmapDSIn1.usiValueIdx	:= 0;
			END_IF

		END_IF
	END_IF
	//DBA B
	IF p_tyNtParamCurr.bUIConvDirRL = FALSE THEN
		IF p_tyMcParamCurr.eDSCommB = McSetCommModSMEMA THEN
			IF p_bDSSMEMABUSRdy = TRUE THEN
				IF p_bDSSMEMABUSGdBrdRdy = TRUE THEN
					tyP0200OpsGen.tyDSCommB.tyBitmapOut.usiValueIdx	:= 1;
				ELSE
					tyP0200OpsGen.tyDSCommB.tyBitmapOut.usiValueIdx	:= 2;
				END_IF
			ELSE
				tyP0200OpsGen.tyDSCommB.tyBitmapOut.usiValueIdx	:= 0;
			END_IF

		ELSIF p_tyMcParamCurr.eDSCommB = McSetCommModHermes THEN
			IF p_bDSHermesBUSRdy = TRUE THEN
				IF p_bDSHermesBUSGdRdy = TRUE THEN
					tyP0200OpsGen.tyDSCommB.tyBitmapOut.usiValueIdx	:= 1;
				ELSE
					tyP0200OpsGen.tyDSCommB.tyBitmapOut.usiValueIdx	:= 2;
				END_IF
			ELSE
				tyP0200OpsGen.tyDSCommB.tyBitmapOut.usiValueIdx	:= 0;
			END_IF

		END_IF
	ELSE
		IF p_tyMcParamCurr.eDSCommB = McSetCommModSMEMA THEN
			IF p_bDSSMEMABUSRdy = TRUE THEN
				IF p_bDSSMEMABUSGdBrdRdy = TRUE THEN
					tyP0200OpsGen.tyDSCommB.tyBitmapOut1.usiValueIdx	:= 1;
				ELSE
					tyP0200OpsGen.tyDSCommB.tyBitmapOut1.usiValueIdx	:= 2;
				END_IF
			ELSE
				tyP0200OpsGen.tyDSCommB.tyBitmapOut1.usiValueIdx	:= 0;
			END_IF

		ELSIF p_tyMcParamCurr.eDSCommB = McSetCommModHermes THEN
			IF p_bDSHermesBUSRdy = TRUE THEN
				IF p_bDSHermesBUSGdRdy = TRUE THEN
					tyP0200OpsGen.tyDSCommB.tyBitmapOut1.usiValueIdx	:= 1;
				ELSE
					tyP0200OpsGen.tyDSCommB.tyBitmapOut1.usiValueIdx	:= 2;
				END_IF
			ELSE
				tyP0200OpsGen.tyDSCommB.tyBitmapOut1.usiValueIdx	:= 0;
			END_IF

		END_IF
	END_IF

	//DSB B
	IF p_tyNtParamCurr.bUIConvDirRL = FALSE THEN
		IF p_tyMcParamCurr.eDSCommB = McSetCommModSMEMA THEN
			IF p_bDSSMEMABDSRdy = TRUE THEN
				tyP0200OpsGen.tyDSCommB.tyBitmapIn.usiValueIdx	:= 1;
			ELSE
				tyP0200OpsGen.tyDSCommB.tyBitmapIn.usiValueIdx	:= 0;
			END_IF

		ELSIF p_tyMcParamCurr.eDSCommB = McSetCommModHermes THEN
			IF p_bDSHermesBDSRdy = TRUE THEN
				IF p_bDSHermesBDSGdRdy = TRUE THEN
					tyP0200OpsGen.tyDSCommB.tyBitmapIn.usiValueIdx	:= 1;
				ELSE
					tyP0200OpsGen.tyDSCommB.tyBitmapIn.usiValueIdx	:= 2;
				END_IF
			ELSE
				tyP0200OpsGen.tyDSCommB.tyBitmapIn.usiValueIdx	:= 0;
			END_IF

		END_IF
	ELSE
		IF p_tyMcParamCurr.eDSCommB = McSetCommModSMEMA THEN
			IF p_bDSSMEMABDSRdy = TRUE THEN
				tyP0200OpsGen.tyDSCommB.tyBitmapIn1.usiValueIdx	:= 1;
			ELSE
				tyP0200OpsGen.tyDSCommB.tyBitmapIn1.usiValueIdx	:= 0;
			END_IF

		ELSIF p_tyMcParamCurr.eDSCommB = McSetCommModHermes THEN
			IF p_bDSHermesBDSRdy = TRUE THEN
				IF p_bDSHermesBDSGdRdy = TRUE THEN
					tyP0200OpsGen.tyDSCommB.tyBitmapIn1.usiValueIdx	:= 1;
				ELSE
					tyP0200OpsGen.tyDSCommB.tyBitmapIn1.usiValueIdx	:= 2;
				END_IF
			ELSE
				tyP0200OpsGen.tyDSCommB.tyBitmapIn1.usiValueIdx	:= 0;
			END_IF

		END_IF
	END_IF

	//Alarm
	IF NOT p_bAlarmErr THEN
		memset(ADR(tyUIAlmData.bAlm) , 0 , SIZEOF(tyUIAlmData.bAlm));
	END_IF

	IF NOT p_bAlarmWarning THEN
		memset(ADR(tyUIAlmData.bWarning) , 0 , SIZEOF(tyUIAlmData.bWarning));
	ELSE
		IF p_bDSHermesAConnected OR p_tyMcParamCurr.eDSCommA = McSetCommModSMEMA THEN
			tyUIAlmData.bWarning[3363] := FALSE;
		END_IF
		IF p_bDSHermesBConnected OR p_tyMcParamCurr.eDSCommB = McSetCommModSMEMA THEN
			tyUIAlmData.bWarning[3531] := FALSE;
		END_IF
	END_IF

	FOR i := 1 TO c_uiP0200TableSize DO
		IF p_bStartupUISettingsLoadDone THEN
			IF p_tyAlarmCurrList[i].eSeverity = AlmSeverityError THEN
				tyUIAlmData.bAlm[p_tyAlarmCurrList[i].udiErrorCode] := p_tyAlarmCurrList[i].bAlm;
			ELSIF p_tyAlarmCurrList[i].eSeverity = AlmSeverityWarning THEN
				tyUIAlmData.bWarning[p_tyAlarmCurrList[i].udiErrorCode] := p_tyAlarmCurrList[i].bWarning;
			END_IF
		END_IF
	END_FOR

	//Magazine Info
	IF p_tyNtParamCurr.bProjAutoRcpPrep AND (p_tyMcParamCurr.bHermesSvyEn OR p_tyNtParamCurr.eCustomerReq = We_Fabricate) THEN
		IF p_ausiSvyMagAccOrder[1] = 10 THEN
			tyP0200OpsGen.tyOps.tyNumMinSltRange.diValue	:= p_diLinkAutoRcpMag1MinSlt;
			tyP0200OpsGen.tyOps.tyNumMaxSltRange.diValue	:= p_diLinkAutoRcpMag1MaxSlt;
			tyP0200OpsGen.tyOps.tyNumPitch.diValue			:= p_diLinkAutoRcpMag1Pitch;
		ELSIF p_ausiSvyMagAccOrder[2] = 10 THEN
			tyP0200OpsGen.tyOps.tyNumMinSltRange.diValue	:= p_diLinkAutoRcpMag2MinSlt;
			tyP0200OpsGen.tyOps.tyNumMaxSltRange.diValue	:= p_diLinkAutoRcpMag2MaxSlt;
			tyP0200OpsGen.tyOps.tyNumPitch.diValue			:= p_diLinkAutoRcpMag2Pitch;
		ELSIF p_ausiSvyMagAccOrder[3] = 10 THEN
			tyP0200OpsGen.tyOps.tyNumMinSltRange.diValue	:= p_diLinkAutoRcpMag3MinSlt;
			tyP0200OpsGen.tyOps.tyNumMaxSltRange.diValue	:= p_diLinkAutoRcpMag3MaxSlt;
			tyP0200OpsGen.tyOps.tyNumPitch.diValue			:= p_diLinkAutoRcpMag3Pitch;
		END_IF
	ELSE //standard
		tyP0200OpsGen.tyOps.tyNumMinSltRange.diValue	:= p_tyProdRcpCurrRcp2.diMinSltValue;
		tyP0200OpsGen.tyOps.tyNumMaxSltRange.diValue	:= p_tyProdRcpCurrRcp2.diMaxSltValue;
		tyP0200OpsGen.tyOps.tyNumPitch.diValue			:= p_tyProdRcpCurrRcp2.diPitch;
	END_IF

	CASE p_tyProdRcpCurrRcp2.usiMcMod OF
		0:
			tyP0200OpsGen.tyOps.tyNumMinSltRangeRear.diValue	:= p_tyProdRcpCurrRcp2.diMinSltValue;
			tyP0200OpsGen.tyOps.tyNumMaxSltRangeRear.diValue	:= p_tyProdRcpCurrRcp2.diMaxSltValue;
			tyP0200OpsGen.tyOps.tyNumPitchRear.diValue			:= p_tyProdRcpCurrRcp2.diPitch;

		1:
			tyP0200OpsGen.tyOps.tyNumMinSltRangeRear.diValue	:= p_tyProdRcpCurrRcp2.diMinSltValueRear;
			tyP0200OpsGen.tyOps.tyNumMaxSltRangeRear.diValue	:= p_tyProdRcpCurrRcp2.diMaxSltValueRear;
			tyP0200OpsGen.tyOps.tyNumPitchRear.diValue			:= p_tyProdRcpCurrRcp2.diPitchRear;

		2:
			tyP0200OpsGen.tyOps.tyNumMinSltRangeRear.diValue	:= p_tyProdRcpCurrRcp2.diMinSltValueRear;
			tyP0200OpsGen.tyOps.tyNumMaxSltRangeRear.diValue	:= p_tyProdRcpCurrRcp2.diMaxSltValueRear;
			tyP0200OpsGen.tyOps.tyNumPitchRear.diValue			:= p_tyProdRcpCurrRcp2.diPitchRear;
		END_CASE

	//Mag1
	IF p_bBuffer1MagPresent = TRUE THEN
		IF p_tyNtParamCurr.eCustomerReq = Siemens AND p_ausiSvyMagAccOrder[1] = 0 AND p_tyMcParamCurr.eDSCommA <> McSetCommModSMEMA
			AND p_tyMcParamCurr.bHermesSvyEn THEN
			tyP0200OpsGen.tyOps.tyNumMag1AvlQty.diValue		:= 0;
			tyP0200OpsGen.tyOps.tyNumMag1TtlSlt.diValue		:= 0;
		ELSE
			tyP0200OpsGen.tyOps.tyNumMag1AvlQty.diValue		:= p_tyBuffer1BffrStat.diTtlBadBrd + p_tyBuffer1BffrStat.diTtlGdBrd;
			tyP0200OpsGen.tyOps.tyNumMag1TtlSlt.diValue		:= p_tyBuffer1BffrStat.diTtlBrdCap;
		END_IF
	ELSE
		tyP0200OpsGen.tyOps.tyNumMag1AvlQty.diValue		:= 0;
		tyP0200OpsGen.tyOps.tyNumMag1TtlSlt.diValue		:= 0;
	END_IF

	//Mag2
	IF p_bBuffer2MagPresent = TRUE THEN
		IF p_tyNtParamCurr.eCustomerReq = Siemens AND p_ausiSvyMagAccOrder[2] = 0 AND p_tyMcParamCurr.eDSCommA <> McSetCommModSMEMA
			AND p_tyMcParamCurr.bHermesSvyEn THEN
			tyP0200OpsGen.tyOps.tyNumMag2AvlQty.diValue		:= 0;
			tyP0200OpsGen.tyOps.tyNumMag2TtlSlt.diValue		:= 0;
		ELSE
			tyP0200OpsGen.tyOps.tyNumMag2AvlQty.diValue		:= p_tyBuffer2BffrStat.diTtlBadBrd + p_tyBuffer2BffrStat.diTtlGdBrd;
			tyP0200OpsGen.tyOps.tyNumMag2TtlSlt.diValue		:= p_tyBuffer2BffrStat.diTtlBrdCap;
		END_IF
	ELSE
		tyP0200OpsGen.tyOps.tyNumMag2AvlQty.diValue		:= 0;
		tyP0200OpsGen.tyOps.tyNumMag2TtlSlt.diValue		:= 0;
	END_IF

	//Mag3
	IF p_bBuffer3MagPresent = TRUE THEN
		IF p_tyNtParamCurr.eCustomerReq = Siemens AND p_ausiSvyMagAccOrder[3] = 0 AND p_tyMcParamCurr.eDSCommA <> McSetCommModSMEMA
			AND p_tyMcParamCurr.bHermesSvyEn THEN
			tyP0200OpsGen.tyOps.tyNumMag3AvlQty.diValue		:= 0;
			tyP0200OpsGen.tyOps.tyNumMag3TtlSlt.diValue		:= 0;
		ELSE
			tyP0200OpsGen.tyOps.tyNumMag3AvlQty.diValue		:= p_tyBuffer3BffrStat.diTtlBadBrd + p_tyBuffer3BffrStat.diTtlGdBrd;
			tyP0200OpsGen.tyOps.tyNumMag3TtlSlt.diValue		:= p_tyBuffer3BffrStat.diTtlBrdCap;
		END_IF
	ELSE
		tyP0200OpsGen.tyOps.tyNumMag3AvlQty.diValue		:= 0;
		tyP0200OpsGen.tyOps.tyNumMag3TtlSlt.diValue		:= 0;
	END_IF

	//Mag4
	IF p_bBuffer4MagPresent = TRUE THEN
		tyP0200OpsGen.tyOps.tyNumMag4AvlQty.diValue		:= p_tyBuffer4BffrStat.diTtlBadBrd + p_tyBuffer4BffrStat.diTtlGdBrd;
		tyP0200OpsGen.tyOps.tyNumMag4TtlSlt.diValue		:= p_tyBuffer4BffrStat.diTtlBrdCap;
	ELSE
		tyP0200OpsGen.tyOps.tyNumMag4AvlQty.diValue		:= 0;
		tyP0200OpsGen.tyOps.tyNumMag4TtlSlt.diValue		:= 0;
	END_IF

END_ACTION
```

#### Act_OptP0200VirtualSMEMA.st
```iecst
ACTION Act_OptP0200VSMEMA:

	//Downstream Virtual SMEMA A
	//Enable / Disable
	IF p_tyNtParamCurr.bUIConvDirRL = FALSE THEN
		IF tyP0200OpsGen.tyOps.tyHotspotDSAVSMEMA.bRtCompl = TRUE THEN
			tyP0200OpsGen.tyOps.tyHotspotDSAVSMEMA.bRtCompl	:= FALSE;

			IF tyP0200OpsGen.tyOps.tyHotspotDSAVSMEMA.bValue = TRUE THEN
				bVSMEMADSAEn	:= TRUE;

				fUIInRtStatOff(ADR(tyP0200OpsGen.tyDSAVSMEMA.tyLyr.uiRtStat));
			ELSE
				tyP0200OpsGen.tyDSAVSMEMA.tyBtnNom.bValue	:= FALSE;

				bVSMEMADSAEn	:= FALSE;

				fUIInRtStatHide(ADR(tyP0200OpsGen.tyDSAVSMEMA.tyLyr.uiRtStat));
			END_IF

		END_IF
	ELSE
		IF tyP0200OpsGen.tyOps.tyHotspotDSAVSMEMA1.bRtCompl = TRUE THEN
			tyP0200OpsGen.tyOps.tyHotspotDSAVSMEMA1.bRtCompl	:= FALSE;

			IF tyP0200OpsGen.tyOps.tyHotspotDSAVSMEMA1.bValue = TRUE THEN
				bVSMEMADSAEn	:= TRUE;

				fUIInRtStatOff(ADR(tyP0200OpsGen.tyDSAVSMEMA1.tyLyr.uiRtStat));
			ELSE
				tyP0200OpsGen.tyDSAVSMEMA1.tyBtnNom.bValue	:= FALSE;

				bVSMEMADSAEn	:= FALSE;

				fUIInRtStatHide(ADR(tyP0200OpsGen.tyDSAVSMEMA1.tyLyr.uiRtStat));
			END_IF

		END_IF
	END_IF

	//Control
	IF p_tyNtParamCurr.bUIConvDirRL = FALSE THEN
		IF tyP0200OpsGen.tyDSAVSMEMA.tyBtnNom.bRtCompl = TRUE THEN
			tyP0200OpsGen.tyDSAVSMEMA.tyBtnNom.bRtCompl	:= FALSE;
		END_IF
	ELSE
		IF tyP0200OpsGen.tyDSAVSMEMA1.tyBtnNom.bRtCompl = TRUE THEN
			tyP0200OpsGen.tyDSAVSMEMA1.tyBtnNom.bRtCompl	:= FALSE;
		END_IF
	END_IF

	//Update
	IF p_tyNtParamCurr.bUIConvDirRL = FALSE THEN
		bVSMEMADSBA	:= tyP0200OpsGen.tyDSAVSMEMA.tyBtnNom.bValue;
	ELSE
		bVSMEMADSBA	:= tyP0200OpsGen.tyDSAVSMEMA1.tyBtnNom.bValue;
	END_IF

	//Downstream Virtual SMEMA B
	//Enable / Disable
	IF p_tyNtParamCurr.bUIConvDirRL = FALSE THEN
		IF tyP0200OpsGen.tyDSCommB.tyHotspotDSBVSMEMA.bRtCompl = TRUE THEN
			tyP0200OpsGen.tyDSCommB.tyHotspotDSBVSMEMA.bRtCompl	:= FALSE;

			IF tyP0200OpsGen.tyDSCommB.tyHotspotDSBVSMEMA.bValue = TRUE THEN
				bVSMEMADSBEn	:= TRUE;

				fUIInRtStatOff(ADR(tyP0200OpsGen.tyDSBVSMEMA.tyLyr.uiRtStat));
			ELSE
				tyP0200OpsGen.tyDSBVSMEMA.tyBtnNom.bValue	:= FALSE;

				bVSMEMADSBEn	:= FALSE;

				fUIInRtStatHide(ADR(tyP0200OpsGen.tyDSBVSMEMA.tyLyr.uiRtStat));
			END_IF

		END_IF
	ELSE
		IF tyP0200OpsGen.tyDSCommB.tyHotspotDSBVSMEMA1.bRtCompl = TRUE THEN
			tyP0200OpsGen.tyDSCommB.tyHotspotDSBVSMEMA1.bRtCompl	:= FALSE;

			IF tyP0200OpsGen.tyDSCommB.tyHotspotDSBVSMEMA1.bValue = TRUE THEN
				bVSMEMADSBEn	:= TRUE;

				fUIInRtStatOff(ADR(tyP0200OpsGen.tyDSBVSMEMA1.tyLyr.uiRtStat));
			ELSE
				tyP0200OpsGen.tyDSBVSMEMA1.tyBtnNom.bValue	:= FALSE;

				bVSMEMADSBEn	:= FALSE;

				fUIInRtStatHide(ADR(tyP0200OpsGen.tyDSBVSMEMA1.tyLyr.uiRtStat));
			END_IF

		END_IF
	END_IF

	//Control
	IF p_tyNtParamCurr.bUIConvDirRL = FALSE THEN
		IF tyP0200OpsGen.tyDSBVSMEMA.tyBtnNom.bRtCompl = TRUE THEN
			tyP0200OpsGen.tyDSBVSMEMA.tyBtnNom.bRtCompl	:= FALSE;
		END_IF
	ELSE
		IF tyP0200OpsGen.tyDSBVSMEMA1.tyBtnNom.bRtCompl = TRUE THEN
			tyP0200OpsGen.tyDSBVSMEMA1.tyBtnNom.bRtCompl	:= FALSE;
		END_IF
	END_IF

	//Update
	IF p_tyNtParamCurr.bUIConvDirRL = FALSE THEN
		bVSMEMADSBB	:= tyP0200OpsGen.tyDSBVSMEMA.tyBtnNom.bValue;
	ELSE
		bVSMEMADSBB	:= tyP0200OpsGen.tyDSBVSMEMA1.tyBtnNom.bValue;
	END_IF

END_ACTION
```

#### Act_OptP0200BarCodeScannerAndOthers.st
```iecst
ACTION Act_OptP0200BarCodeScannerAndOthers:

	//Mask

	IF p_bBuffer1MagPresent = FALSE
		AND p_bBuffer2MagPresent = FALSE
		AND  p_bBuffer3MagPresent = FALSE
		AND p_bBuffer4MagPresent = FALSE
		THEN
		fUIInRtStatHide(ADR(tyP0200OpsGen.tyOps.tyBtnBarCodeScan.uiMaskRtStat));
		fbLMCfbTm(IN:= FALSE); //Reset LMC feedback timer
	ELSE
		fUIInRtStatOff(ADR(tyP0200OpsGen.tyOps.tyBtnBarCodeScan.uiMaskRtStat));
		fUIInRtStatHide(ADR(tyP0200OpsGen.tyBarCodeScan.tyLyr.uiRtStat));
	END_IF

	//BarCode Scanner Pressed
	IF tyP0200OpsGen.tyOps.tyBtnBarCodeScan.bRtCompl = TRUE THEN
		tyP0200OpsGen.tyOps.tyBtnBarCodeScan.bRtCompl := FALSE;

		tyP0200OpsGen.tyBarCodeScan.tyStringBarCode.sValue := '';
		tyP0200OpsGen.tyBarCodeScan.tyStringWorkOrder.sValue := '';
		fUIInRtStatOff(ADR(tyP0200OpsGen.tyBarCodeScan.tyLyr.uiRtStat));
	END_IF

	//String Check
	IF LEN(tyP0200OpsGen.tyBarCodeScan.tyStringBarCode.sValue) > 15 THEN
		p_tyC0008MsgBox ACCESS (ADR(tyP0200OpsGen.tyMsgBoxBarCode));
	END_IF

	IF tyP0200OpsGen.tyMsgBoxBarCode.tyBtnNo.bRtCompl = TRUE THEN
		tyP0200OpsGen.tyMsgBoxBarCode.tyBtnNo.bRtCompl 	:= FALSE;
		tyP0200OpsGen.tyMsgBoxBarCode.tyBtnNo.bValue	:= FALSE;

		p_tyC0008MsgBox ACCESS ADR(tyP0200OpsGen.tyMsgBoxHide);
		tyP0200OpsGen.tyBarCodeScan.tyStringBarCode.sValue	:= '';
		tyP0200OpsGen.tyBarCodeScan.tyStringWorkOrder.sValue := '';
	END_IF

	//Trolley Unlock
	//ops control
END_ACTION
```

#### Act_OptP0200BarCodeChgRcp.st
```iecst
ACTION Act_OptP0200BarCodeChgRcp:
	//Work order
	tyP0200OpsGen.tyBarCodeScan.tyStringWorkOrder.uiRtStat := NOT(p_tyNtParamCurr.bProjWorkOrderOPCUA);

	IF p_tyNtParamCurr.bBCodeScannerPrep THEN

		CASE p_tyNtParamCurr.eScannerType OF

			RS232:

				IF tyP0200OpsGen.tyBarCodeScan.tyLyr.uiRtStat.0 = FALSE THEN

					eFrmAct	:= FrmActFullReadUntilValid;

					IF p_eFrmStat = FrmActFullReadUntilValid AND p_eFrmStatus = Done THEN

						IF p_bFrmMsgRdValid = TRUE THEN
							eFrmAct := FrmActIdle;
							IF p_tyNtParamCurr.bProjWorkOrderOPCUA THEN
								tyP0200OpsGen.tyBarCodeScan.tyStringWorkOrder.sValue := LEFT(p_sFrmMsgRd,FIND(p_sFrmMsgRd,'@')-1);
								tyP0200OpsGen.tyBarCodeScan.tyStringBarCode.sValue	:= DELETE(p_sFrmMsgRd,LEN(tyP0200OpsGen.tyBarCodeScan.tyStringWorkOrder.sValue)+1,1);
							ELSE
								tyP0200OpsGen.tyBarCodeScan.tyStringBarCode.sValue	:= p_sFrmMsgRd;
							END_IF

						ELSE
							eFrmAct := FrmActIdle;
							tyP0200OpsGen.tyBarCodeScan.tyStringBarCode.sValue	:= '';
						END_IF

					END_IF

				END_IF

			USB:

				bUSBRun := tyP0200OpsGen.tyBarCodeScan.tyLyr.uiRtStat.0 = FALSE;

				IF tyP0200OpsGen.tyBarCodeScan.tyLyr.uiRtStat.0 = FALSE THEN // Can Continue Reading Data.

						 IF p_eUSBRdrStatus<>Error THEN

							CASE usiUSBBarcodeStep OF

								0:

									eUSBRdrAct	:= USBRdrActDetectDev;

									IF p_eUSBRdrStat = USBRdrActDetectDev AND p_eUSBRdrStatus = Done THEN

										eUSBRdrAct	:= USBRdrActIdle;

										usiUSBBarcodeStep := 1;

									END_IF

								1:

									eUSBRdrAct	:= USBRdrActRead;

									IF p_eUSBRdrStat = USBRdrActRead AND p_eUSBRdrStatus = Done THEN

										eUSBRdrAct	:= USBRdrActIdle;

										tyP0200OpsGen.tyBarCodeScan.tyStringBarCode.sValue := p_sUSBRdrBarcodeOut;

										usiUSBBarcodeStep := 0;

									END_IF
							END_CASE

						END_IF

				ELSE // layer hide
					eUSBRdrAct	:= USBRdrActIdle;
					usiUSBBarcodeStep := 0;

				END_IF
		END_CASE

	END_IF

	IF tyP0200OpsGen.tyBarCodeScan.tyBtnOK.bRtCompl THEN

		CASE usiChgRcpStep OF

			0:
				tyProdRcpInfoIn.sRcpNm		:= 	tyP0200OpsGen.tyBarCodeScan.tyStringBarCode.sValue;

				eProdRcpAct					:=  ProdRcpActLoadRcp;

				IF p_eProdRcpStat = ProdRcpActLoadRcp AND p_eProdRcpStatus = Done THEN

					eProdRcpAct	:= ProdRcpActIdle;

					IF p_bProdRcpNmEmpty = TRUE OR p_bProdRcpNmNotExist = TRUE THEN

						usiChgRcpStep	:= 1;

					ELSE
						//Update UI Current Recipe
						tyP0400ProdSel.tyProdSel.tyStringRecipeNm.sValue	:= p_tyProdRcpCurrRcp0.sRcpNm;
						tyP0400ProdSel.tyProdSel.tyNumProdWidth.diValue		:= p_tyProdRcpCurrRcp0.diWidthInUM;

						tyProdRcpCurrRcpWr	:= p_tyProdRcpCurrRcp0;

						usiChgRcpStep	:= 2;

					END_IF

				ELSIF p_eProdRcpStatus = Error THEN

					usiChgRcpStep	:= 3;

				END_IF

			1:
				//Message Name Not Found
				p_tyC0008MsgBox ACCESS ADR(tyP0200OpsGen.tyMsgBoxSelRcpNoNm);

				IF tyP0200OpsGen.tyMsgBoxSelRcpNoNm.tyBtnNo.bRtCompl = TRUE THEN
					tyP0200OpsGen.tyMsgBoxSelRcpNoNm.tyBtnNo.bRtCompl	:= FALSE;
					tyP0200OpsGen.tyMsgBoxSelRcpNoNm.tyBtnNo.bValue		:= FALSE;

					p_tyC0008MsgBox ACCESS ADR(tyP0200OpsGen.tyMsgBoxHide);

					tyP0200OpsGen.tyBarCodeScan.tyBtnOK.bRtCompl := FALSE;
					tyP0200OpsGen.tyBarCodeScan.tyBtnOK.bValue	 := FALSE;

					usiChgRcpStep	:= 0;
				END_IF

			2: 	IF p_tyMcParamCurr.bLFEn AND p_tyNtParamCurr.bLFPrep AND (p_tyMcParamCurr.eDSCommA = McSetCommModSMEMA AND p_tyMcParamCurr.eDSCommB = McSetCommModSMEMA) THEN

					p_tyC0008MsgBox ACCESS ADR(tyP0200OpsGen.tyMsgBoxGoToLFCtrlAsk);

					IF tyP0200OpsGen.tyMsgBoxGoToLFCtrlAsk.tyBtnYes.bRtCompl = TRUE THEN
						tyP0200OpsGen.tyMsgBoxGoToLFCtrlAsk.tyBtnYes.bRtCompl	:= FALSE;
						tyP0200OpsGen.tyMsgBoxGoToLFCtrlAsk.tyBtnYes.bValue		:= FALSE;

						eChgPage	:= UIP0700LFCtrl;

						//Start Operation
						tyCommon.tyMain.tyBtnStart.bRtCompl	:= TRUE;

						usiChgRcpStep	:= 3;

						p_tyC0008MsgBox ACCESS ADR(tyP0200OpsGen.tyMsgBoxHide);

					ELSIF tyP0200OpsGen.tyMsgBoxGoToLFCtrlAsk.tyBtnNo.bRtCompl = TRUE THEN

						tyP0200OpsGen.tyMsgBoxGoToLFCtrlAsk.tyBtnNo.bRtCompl	:= FALSE;
						tyP0200OpsGen.tyMsgBoxGoToLFCtrlAsk.tyBtnNo.bValue		:= FALSE;

						p_tyC0008MsgBox ACCESS ADR(tyP1021McSetGen.tyMsgBoxHide);

						usiChgRcpStep	:= 3;

					END_IF
				ELSE
					usiChgRcpStep	:= 3;
				END_IF

			3:
				//Reset

				tyP0200OpsGen.tyBarCodeScan.tyBtnOK.bRtCompl	:= FALSE;
				tyP0200OpsGen.tyBarCodeScan.tyBtnOK.bValue		:= FALSE;
				tyP0200OpsGen.tyOps.tyBtnBarCodeScan.bValue		:= FALSE;

				fUIInRtStatHide(ADR(tyP0200OpsGen.tyBarCodeScan.tyLyr.uiRtStat));

				usiChgRcpStep	:= 0;
				bBlkOpsTravLif := FALSE; //unblock operation

		END_CASE

	ELSIF  tyP0200OpsGen.tyBarCodeScan.tyBtnCancel.bRtCompl THEN

		tyP0200OpsGen.tyBarCodeScan.tyBtnCancel.bRtCompl		:= FALSE;
		tyP0200OpsGen.tyBarCodeScan.tyBtnCancel.bValue			:= FALSE;
		tyP0200OpsGen.tyOps.tyBtnBarCodeScan.bValue				:= FALSE;

		fUIInRtStatHide(ADR(tyP0200OpsGen.tyBarCodeScan.tyLyr.uiRtStat));

	END_IF

	// Error Reset
	IF p_tyNtParamCurr.eScannerType = USB THEN
		IF p_eUSBRdrStatus = Error THEN
			usiUSBBarcodeStep	:= 0;
			tyP0200OpsGen.tyBarCodeScan.tyStringBarCode.sValue := '';
		END_IF
	END_IF

END_ACTION
```

#### Act_OptP0200Keypad.st
```iecst
ACTION Act_OptP0200Keypad:

	IF fUIOutRtStatTPIsOpen(ADR(tyP0200OpsGen.tyBarCodeScan.tyStringBarCode.uiRtStat)) = TRUE THEN
		tyProperty.tyKeypad.tyStringTitle.sKeypadTitle			:= tyP0200OpsGen.tyBarCodeScan.tyStringBarCode.sKeypadTitle;
	END_IF

END_ACTION
```

#### Act_OptP0200WorkOrderToLMC.st
```iecst
ACTION Act_OptP0200WorkOrderToLMC:
	IF p_tyNtParamCurr.bProjWorkOrderOPCUA AND
		tyP0200OpsGen.tyBarCodeScan.tyStringWorkOrder.sValue <> '' THEN
		tyTagNm.sWorkOrder := tyP0200OpsGen.tyBarCodeScan.tyStringWorkOrder.sValue;

		IF (bMag1Active OR bMag2Active )AND (p_tyBuffer1BffrStat.bBffrMty OR p_bBuffer1MagPresent = FALSE)
			AND (p_tyBuffer2BffrStat.bBffrMty OR p_bBuffer2MagPresent = FALSE) AND fbLMCfbTm.Q  = FALSE THEN
			p_tyC0008MsgBox ACCESS ADR(tyP0200OpsGen.tyMsgBoxWOFinished); //"Work Order Done. Wait for LMC complete."
			bBlkOpsTravLif := TRUE; // block operation to next magazine
			fbLMCfbTm(IN:= TRUE,PT:= DINT_TO_TIME(p_tyMcParamCurr.diLMCfbTmInMS)); //wait for LMC done

			IF tyTagNm.uiQuantities = diMag1TtSlt + diMag2TtSlt THEN //LMC done
				fbLMCfbTm(IN:= FALSE);
				bMag1Active := FALSE;
				bMag2Active := FALSE;
				tyP0200OpsGen.tyBarCodeScan.tyStringWorkOrder.sValue := '';
				p_tyC0008MsgBox ACCESS ADR(tyP0200OpsGen.tyMsgBoxLMCCompl); //LMC completed. Scan for new Work Order.
			END_IF

			//		IF bMag1Active AND p_tyBuffer1BffrStat.bBffrMty AND fbLMCfbTm.Q  = FALSE THEN
			//			p_tyC0008MsgBox ACCESS ADR(tyP0200OpsGen.tyMsgBoxWOFinished); //"Work Order Done. Wait for LMC complete."
			//			bBlkOpsTravLif := TRUE; // block operation to next magazine
			//			fbLMCfbTm(IN:= TRUE,PT:= DINT_TO_TIME(p_tyMcParamCurr.diLMCfbTmInMS)); //wait for LMC done
			//
			//			IF tyTagNm.uiQuantities = p_tyBuffer1BffrStat.diTtlBrdCap THEN //LMC done
			//				tyP0200OpsGen.tyBarCodeScan.tyStringWorkOrder.sValue := '';
			//				p_tyC0008MsgBox ACCESS ADR(tyP0200OpsGen.tyMsgBoxLMCCompl); //LMC completed. Scan for new Work Order.
			//			END_IF
			//
			//		ELSIF bMag2Active AND p_tyBuffer2BffrStat.bBffrMty  AND fbLMCfbTm.Q  = FALSE THEN
			//			p_tyC0008MsgBox ACCESS ADR(tyP0200OpsGen.tyMsgBoxWOFinished); //"Work Order Done. Wait for LMC complete."
			//			bBlkOpsTravLif := TRUE; // block operation to next magazine
			//			fbLMCfbTm(IN:= TRUE,PT:= DINT_TO_TIME(p_tyMcParamCurr.diLMCfbTmInMS)); //wait for LMC done
			//
			//			IF tyTagNm.uiQuantities = p_tyBuffer2BffrStat.diTtlBrdCap THEN //LMC done
			//				tyP0200OpsGen.tyBarCodeScan.tyStringWorkOrder.sValue := '';
			//				p_tyC0008MsgBox ACCESS ADR(tyP0200OpsGen.tyMsgBoxLMCCompl);
			//			END_IF

		ELSIF fbLMCfbTm.Q THEN
			p_tyC0008MsgBox ACCESS ADR(tyP0200OpsGen.tyMsgBoxLMCFail);//No Feedback From LMC.
		//	iTtWorkOrderSlt := DINT_TO_UINT(diMag1TtSlt) + DINT_TO_UINT(diMag2TtSlt);
			diTtWorkOrderSlt := diMag1TtSlt + diMag2TtSlt;
			string1 := DINT_TO_STRING(diTtWorkOrderSlt);
			string2 := UINT_TO_STRING(tyTagNm.uiQuantities);
			tyTagNm.sLogMessage := CONCAT('No Exact Quantities Received. Total ',string1);
			tyTagNm.sLogMessage := CONCAT(tyTagNm.sLogMessage,' boards, received ');
			tyTagNm.sLogMessage := CONCAT(tyTagNm.sLogMessage, string2);
			tyTagNm.sLogMessage := CONCAT(tyTagNm.sLogMessage,' boards.');

			tyTagNm.diTotalBrd := diTtWorkOrderSlt;
			tyP0200OpsGen.tyMsgBoxLMCFail.tyTxtWO_sLogMessage.uiRtStat := FALSE;
			tyP0200OpsGen.tyMsgBoxLMCFail.tyTxtWO_sLogMessage.sValue := tyTagNm.sLogMessage;

		END_IF
		//
		//		IF tyTagNm.uiQuantities >0 THEN
		//			IF bInitQuanValue = FALSE THEN
		//				bInitQuanValue := TRUE;
		//				uiBrdOutCntr := tyTagNm.uiQuantities;
		//			END_IF
		//			tyTagNm.bProcess := TRUE;
		//		ELSE
		//			bInitQuanValue := FALSE;
		//			uiBrdOutCntr := 0;
		//			tyTagNm.bProcess := FALSE;
		//		END_IF

	ELSE
		bBlkOpsTravLif := FALSE;
		bMag1Active := FALSE;
		bMag2Active := FALSE;
		fbLMCfbTm(IN:= FALSE);
	END_IF

	//	IF EDGEPOS(uiBrdOutCntr = 0) AND tyTagNm.uiQuantities >0 THEN //LMC in process
	//		p_tyC0008MsgBox ACCESS ADR(tyP0200OpsGen.tyMsgBoxWOFinished);
	//	END_IF
	//
	//	IF EDGEPOS(p_bOpsTravLifLDExitBrd) AND uiBrdOutCntr <> 0 THEN
	//		uiBrdOutCntr := uiBrdOutCntr -1;
	//	END_IF

	//======================== Message Box btn ==================================
	//Close msgbox (tyMsgBoxWOFinished)
	IF tyP0200OpsGen.tyMsgBoxWOFinished.tyBtnNo.bRtCompl = TRUE THEN
		tyP0200OpsGen.tyMsgBoxWOFinished.tyBtnNo.bRtCompl	:= FALSE;
		tyP0200OpsGen.tyMsgBoxWOFinished.tyBtnNo.bValue		:= FALSE;

		p_tyC0008MsgBox ACCESS ADR(tyP0200OpsGen.tyMsgBoxHide);
	END_IF

	//(tyMsgBoxLMCFail)
	IF tyP0200OpsGen.tyMsgBoxLMCFail.tyBtnNo.bRtCompl THEN //ok
		tyP0200OpsGen.tyMsgBoxLMCFail.tyBtnNo.bRtCompl := FALSE;
		tyP0200OpsGen.tyMsgBoxLMCFail.tyBtnNo.bValue := FALSE;
		p_tyC0008MsgBox ACCESS ADR(tyP0200OpsGen.tyMsgBoxHide);

		bBlkOpsTravLif := FALSE;
		bMag1Active := FALSE;
		bMag2Active := FALSE;
		fbLMCfbTm(IN:= FALSE);
		tyTagNm.uiQuantities := 0; //Reset quantities from LMC
		tyP0200OpsGen.tyMsgBoxLMCFail.tyTxtWO_sLogMessage.uiRtStat := TRUE;

	ELSIF tyP0200OpsGen.tyMsgBoxLMCFail.tyBtnYes.bRtCompl THEN //scan //hide(true)
		tyP0200OpsGen.tyMsgBoxLMCFail.tyBtnYes.bRtCompl := FALSE;
		tyP0200OpsGen.tyMsgBoxLMCFail.tyBtnYes.bValue 	:= FALSE;
		p_tyC0008MsgBox ACCESS ADR(tyP0200OpsGen.tyMsgBoxHide);

		tyP0200OpsGen.tyBarCodeScan.tyStringBarCode.sValue := '';
		tyP0200OpsGen.tyBarCodeScan.tyStringWorkOrder.sValue := '';
		fUIInRtStatOff(ADR(tyP0200OpsGen.tyBarCodeScan.tyLyr.uiRtStat));

	END_IF

	//(tyMsgBoxLMCCompl)
	IF tyP0200OpsGen.tyMsgBoxLMCCompl.tyBtnNo.bRtCompl THEN //ok
		tyP0200OpsGen.tyMsgBoxLMCCompl.tyBtnNo.bRtCompl := FALSE;
		tyP0200OpsGen.tyMsgBoxLMCCompl.tyBtnNo.bValue	:= FALSE;
		p_tyC0008MsgBox ACCESS ADR(tyP0200OpsGen.tyMsgBoxHide);

		bBlkOpsTravLif := FALSE;
		bMag1Active := FALSE;
		bMag2Active := FALSE;
		fbLMCfbTm(IN:= FALSE);

		tyP0200OpsGen.tyBarCodeScan.tyStringBarCode.sValue := '';
		tyP0200OpsGen.tyBarCodeScan.tyStringWorkOrder.sValue := '';
		tyTagNm.uiQuantities := 0; //Reset quantities from LMC
		fUIInRtStatOff(ADR(tyP0200OpsGen.tyBarCodeScan.tyLyr.uiRtStat));

	ELSIF tyP0200OpsGen.tyMsgBoxLMCCompl.tyBtnYes.bRtCompl THEN //N/A

	END_IF
	//======================== ##==================================

	//Determine active magazine
	IF p_eOpsTravLifPosGo = TravLifLDPosUS1 THEN
		bMag1Active := TRUE;
	ELSIF p_eOpsTravLifPosGo = TravLifLDPosUS2 THEN
		bMag2Active := TRUE;
	END_IF

	IF p_bBuffer1MagPresent = FALSE THEN
		diMag1TtSlt := 0;
	ELSE
		diMag1TtSlt := p_tyBuffer1BffrStat.diTtlBrdCap;
	END_IF
	IF p_bBuffer2MagPresent = FALSE THEN
		diMag2TtSlt := 0;
	ELSE
		diMag2TtSlt := p_tyBuffer2BffrStat.diTtlBrdCap;
	END_IF

	//Error
	IF p_bOpsRun = FALSE THEN
		p_tyC0008MsgBox ACCESS ADR(tyP0200OpsGen.tyMsgBoxHide);
		IF p_bBuffer1MagRemoved THEN
			tyTagNm.sLogMessage := 'Loader Magazine 1 had removed.';
		ELSIF p_bBuffer2MagRemoved THEN
			tyTagNm.sLogMessage := 'Loader Magazine 2 had removed.';
		ELSIF p_bAlarmErr THEN
			tyTagNm.sLogMessage := 'Loader Alarm activated.';
		END_IF
	END_IF

END_ACTION
```

#### Act_EntP0201Disp.st
```iecst
ACTION Act_EntP0201Disp:

	//Access Address
	p_tyC0004Navi ACCESS ADR(tyP0201OpsTravLifter.tyNaviBack);

	p_tyC0005Main ACCESS ADR(tyCommon.tyMain);

	p_tyC0007Notif ACCESS ADR(tyCommon.tyNotif);

	p_tyC0008MsgBox ACCESS ADR(tyP0201OpsTravLifter.tyMsgBoxHide);

	p_tyC0009Info ACCESS ADR(tyCommon.tyInfo);

	p_tyC0011RcpPopUp ACCESS ADR(tyP0201OpsTravLifter.tyRcpPopUp);

	p_tyP0201OpsTravLif ACCESS ADR(tyP0201OpsTravLifter.tyOps);
	p_tyP0201TravLifIOMonitor ACCESS ADR(tyP0201OpsTravLifter.tyIOMonitor);
	p_tyP0201TravLifBypsInitConv ACCESS ADR(tyP0201OpsTravLifter.tyBypsInitConv);
	p_tyP0201Param ACCESS ADR(tyP0201OpsTravLifter.tyParam);

	p_tyP0201OpsQueryBoardInfo ACCESS ADR(tyP0201OpsTravLifter.tyQueryBoardInfo);//new for Hermes 1.3
	p_tyP0201OpsCurrWorkOrder ACCESS ADR(tyP0201OpsTravLifter.tyCurrWorkOrderInfo);//new for Hermes 1.3
	p_tyP0201OpsQueryWorkOrder ACCESS ADR(tyP0201OpsTravLifter.tyQueryWorkOrderInfo);//new for Hermes 1.3
	p_tyP0201OpsBarcodeScanner ACCESS ADR(tyP0201OpsTravLifter.tyBarcodeScanner);//new for Hermes 1.3

	//Display
	fUIInRtStatHide(ADR(tyP0201OpsTravLifter.tyIOMonitor.tyLyr.uiRtStat));
	fUIInRtStatHide(ADR(tyP0201OpsTravLifter.tyParam.tyLyr.uiRtStat));

	tyP0201OpsTravLifter.tyOps.tyBtnChgParam.uiRtStat.0	:= NOT(p_tyMcParamCurr.bChgParamEn);
	tyP0201OpsTravLifter.tyParam.tyNumMaxSlt.diValueMax	:= p_tyMagRcpCurrRcp.diTtlSlt;

	IF p_tyNtParamCurr.eProjMag = LDMagQuadruple THEN
		fUIInRtStatOff(ADR(tyP0201OpsTravLifter.tyOps.tyLyrProdRear.uiRtStat));
	END_IF

	tyP0201OpsTravLifter.tyParam.tyNumMaxSlt.diValueMax	:= p_tyMagRcpCurrRcp.diTtlSlt;

END_ACTION
```

#### Act_OptP0201BarcodeScanner.st
```iecst
ACTION Act_OptP0201BarcodeScanner:

    //Reset bValue
	IF tyP0201OpsTravLifter.tyBarcodeScanner.tyBtnTop.bRtCompl = TRUE  THEN
		tyP0201OpsTravLifter.tyBarcodeScanner.tyBtnTop.bRtCompl := FALSE;

		tyP0201OpsTravLifter.tyBarcodeScanner.tyBtnBottom.bValue := FALSE;
		tyP0201OpsTravLifter.tyBarcodeScanner.tyBtnMagazine.bValue := FALSE;
		tyP0201OpsTravLifter.tyBarcodeScanner.tyBtnPCB.bValue := FALSE;

	END_IF

	IF tyP0201OpsTravLifter.tyBarcodeScanner.tyBtnBottom.bRtCompl = TRUE  THEN
		tyP0201OpsTravLifter.tyBarcodeScanner.tyBtnBottom.bRtCompl := FALSE;

		tyP0201OpsTravLifter.tyBarcodeScanner.tyBtnTop.bValue := FALSE;
		tyP0201OpsTravLifter.tyBarcodeScanner.tyBtnMagazine.bValue := FALSE;
		tyP0201OpsTravLifter.tyBarcodeScanner.tyBtnPCB.bValue := FALSE;
	END_IF

	IF tyP0201OpsTravLifter.tyBarcodeScanner.tyBtnMagazine.bRtCompl = TRUE  THEN
		tyP0201OpsTravLifter.tyBarcodeScanner.tyBtnMagazine.bRtCompl := FALSE;

		tyP0201OpsTravLifter.tyBarcodeScanner.tyBtnTop.bValue := FALSE;
		tyP0201OpsTravLifter.tyBarcodeScanner.tyBtnBottom.bValue := FALSE;
		tyP0201OpsTravLifter.tyBarcodeScanner.tyBtnPCB.bValue := FALSE;
	END_IF

	IF tyP0201OpsTravLifter.tyBarcodeScanner.tyBtnPCB.bRtCompl = TRUE  THEN
		tyP0201OpsTravLifter.tyBarcodeScanner.tyBtnPCB.bRtCompl := FALSE;

		tyP0201OpsTravLifter.tyBarcodeScanner.tyBtnTop.bValue := FALSE;
		tyP0201OpsTravLifter.tyBarcodeScanner.tyBtnBottom.bValue := FALSE;
		tyP0201OpsTravLifter.tyBarcodeScanner.tyBtnMagazine.bValue := FALSE;
	END_IF

	//Top Barcode
	IF EDGEPOS (tyP0201OpsTravLifter.tyBarcodeScanner.tyBtnTop.bValue = TRUE) THEN
		tyP0201OpsTravLifter.tyBarcodeScanner.tyStringBarcode.sValue := tyP0201OpsTravLifter.tyBarcodeScanner.tyStringTopBarcodeBK.sValue;
	END_IF

	IF EDGENEG (tyP0201OpsTravLifter.tyBarcodeScanner.tyBtnTop.bValue = TRUE) THEN
		tyP0201OpsTravLifter.tyBarcodeScanner.tyStringTopBarcodeBK.sValue := tyP0201OpsTravLifter.tyBarcodeScanner.tyStringTopBarcode.sValue;
	END_IF

	IF tyP0201OpsTravLifter.tyBarcodeScanner.tyBtnTop.bValue = TRUE AND tyP0201OpsTravLifter.tyBarcodeScanner.tyBtnBottom.bValue = FALSE  THEN
		tyP0201OpsTravLifter.tyBarcodeScanner.tyStringTopBarcode.sValue := tyP0201OpsTravLifter.tyBarcodeScanner.tyStringBarcode.sValue;
	END_IF

	//Bottom Barcode
	IF EDGEPOS (tyP0201OpsTravLifter.tyBarcodeScanner.tyBtnBottom.bValue = TRUE) THEN
		tyP0201OpsTravLifter.tyBarcodeScanner.tyStringBarcode.sValue := tyP0201OpsTravLifter.tyBarcodeScanner.tyStringBottomBarcodeBK.sValue;
	END_IF

	IF EDGENEG (tyP0201OpsTravLifter.tyBarcodeScanner.tyBtnBottom.bValue = TRUE) THEN
		tyP0201OpsTravLifter.tyBarcodeScanner.tyStringBottomBarcodeBK.sValue := tyP0201OpsTravLifter.tyBarcodeScanner.tyStringBottomBarcode.sValue;
	END_IF

	IF tyP0201OpsTravLifter.tyBarcodeScanner.tyBtnBottom.bValue = TRUE AND tyP0201OpsTravLifter.tyBarcodeScanner.tyBtnTop.bValue = FALSE THEN
		tyP0201OpsTravLifter.tyBarcodeScanner.tyStringBottomBarcode.sValue := tyP0201OpsTravLifter.tyBarcodeScanner.tyStringBarcode.sValue;
	END_IF

	//Magazine Barcode
	IF EDGEPOS (tyP0201OpsTravLifter.tyBarcodeScanner.tyBtnMagazine.bValue = TRUE) THEN
		tyP0201OpsTravLifter.tyBarcodeScanner.tyStringBarcode.sValue := tyP0201OpsTravLifter.tyBarcodeScanner.tyStringMagazineBarcodeBK.sValue;
	END_IF

	IF EDGENEG (tyP0201OpsTravLifter.tyBarcodeScanner.tyBtnMagazine.bValue = TRUE) THEN
		tyP0201OpsTravLifter.tyBarcodeScanner.tyStringMagazineBarcodeBK.sValue := tyP0201OpsTravLifter.tyBarcodeScanner.tyStringMagazineBarcode.sValue;
	END_IF

	IF tyP0201OpsTravLifter.tyBarcodeScanner.tyBtnMagazine.bValue = TRUE AND tyP0201OpsTravLifter.tyBarcodeScanner.tyBtnPCB.bValue = FALSE THEN
		tyP0201OpsTravLifter.tyBarcodeScanner.tyStringMagazineBarcode.sValue := tyP0201OpsTravLifter.tyBarcodeScanner.tyStringBarcode.sValue;
	END_IF

	//PCB Barcode
	IF EDGEPOS (tyP0201OpsTravLifter.tyBarcodeScanner.tyBtnPCB.bValue = TRUE) THEN
		tyP0201OpsTravLifter.tyBarcodeScanner.tyStringBarcode.sValue := tyP0201OpsTravLifter.tyBarcodeScanner.tyStringPCBBarcodeBK.sValue;
	END_IF

	IF EDGENEG (tyP0201OpsTravLifter.tyBarcodeScanner.tyBtnPCB.bValue = TRUE) THEN
		tyP0201OpsTravLifter.tyBarcodeScanner.tyStringPCBBarcodeBK.sValue := tyP0201OpsTravLifter.tyBarcodeScanner.tyStringPCBBarcode.sValue;
	END_IF

	IF tyP0201OpsTravLifter.tyBarcodeScanner.tyBtnPCB.bValue = TRUE AND tyP0201OpsTravLifter.tyBarcodeScanner.tyBtnMagazine.bValue = FALSE THEN
		tyP0201OpsTravLifter.tyBarcodeScanner.tyStringPCBBarcode.sValue := tyP0201OpsTravLifter.tyBarcodeScanner.tyStringBarcode.sValue;
	END_IF

	//Reset to dummy
	IF tyP0201OpsTravLifter.tyBarcodeScanner.tyBtnTop.bValue = FALSE AND  tyP0201OpsTravLifter.tyBarcodeScanner.tyBtnBottom.bValue = FALSE AND tyP0201OpsTravLifter.tyBarcodeScanner.tyBtnMagazine.bValue = FALSE AND tyP0201OpsTravLifter.tyBarcodeScanner.tyBtnPCB.bValue = FALSE THEN
		tyP0201OpsTravLifter.tyBarcodeScanner.tyStringBarcode.sValue := '';
	END_IF

	//Press OK
	IF	tyP0201OpsTravLifter.tyBarcodeScanner.tyBtnOk.bRtCompl = TRUE THEN

		fUIInRtStatHide(ADR(tyP0201OpsTravLifter.tyBarcodeScanner.tyLyr.uiRtStat)); //hide
		IF tyP0201OpsTravLifter.tyQueryBoardInfo.tyBtnQueryBoardInfo.bValue THEN
			fUIInRtStatOff(ADR(tyP0201OpsTravLifter.tyQueryBoardInfo.tyLyr.uiRtStat)); //show
			tyP0201OpsTravLifter.tyQueryBoardInfo.tyStringTopBarcode.sValue := tyP0201OpsTravLifter.tyBarcodeScanner.tyStringTopBarcode.sValue;
			tyP0201OpsTravLifter.tyQueryBoardInfo.tyStringBottomBarcode.sValue := tyP0201OpsTravLifter.tyBarcodeScanner.tyStringBottomBarcode.sValue;
		ELSIF tyP0201OpsTravLifter.tyCurrWorkOrderInfo.tyBtnQueryWorkOrderInfo.bValue THEN
			fUIInRtStatOff(ADR(tyP0201OpsTravLifter.tyQueryWorkOrderInfo.tyLyr.uiRtStat)); //show
			tyP0201OpsTravLifter.tyQueryWorkOrderInfo.tyStringMagazineId.sValue := tyP0201OpsTravLifter.tyBarcodeScanner.tyStringMagazineBarcode.sValue;
			tyP0201OpsTravLifter.tyQueryWorkOrderInfo.tyStringBarcode.sValue := tyP0201OpsTravLifter.tyBarcodeScanner.tyStringPCBBarcode.sValue;
		END_IF

		tyP0201OpsTravLifter.tyQueryBoardInfo.tyBtnBarcodeScanner.bValue := FALSE;
		tyP0201OpsTravLifter.tyQueryWorkOrderInfo.tyBtnBarcodeScanner.bValue := FALSE;

		tyP0201OpsTravLifter.tyBarcodeScanner.tyBtnOk.bRtCompl := FALSE;
		tyP0201OpsTravLifter.tyBarcodeScanner.tyBtnOk.bValue := FALSE;
		tyP0201OpsTravLifter.tyBarcodeScanner.tyBtnTop.bValue := FALSE;
		tyP0201OpsTravLifter.tyBarcodeScanner.tyBtnBottom.bValue := FALSE;
		tyP0201OpsTravLifter.tyBarcodeScanner.tyBtnMagazine.bValue := FALSE;
		tyP0201OpsTravLifter.tyBarcodeScanner.tyBtnPCB.bValue := FALSE;
		tyP0201OpsTravLifter.tyBarcodeScanner.tyStringBarcode.sValue :='';
		tyP0201OpsTravLifter.tyBarcodeScanner.tyStringTopBarcode.sValue :='';
		tyP0201OpsTravLifter.tyBarcodeScanner.tyStringTopBarcodeBK.sValue :='';
		tyP0201OpsTravLifter.tyBarcodeScanner.tyStringBottomBarcode.sValue :='';
		tyP0201OpsTravLifter.tyBarcodeScanner.tyStringBottomBarcodeBK.sValue :='';
		tyP0201OpsTravLifter.tyBarcodeScanner.tyStringMagazineBarcode.sValue :='';
		tyP0201OpsTravLifter.tyBarcodeScanner.tyStringMagazineBarcodeBK.sValue :='';
		tyP0201OpsTravLifter.tyBarcodeScanner.tyStringPCBBarcode.sValue :='';
		tyP0201OpsTravLifter.tyBarcodeScanner.tyStringPCBBarcodeBK.sValue :='';

	END_IF

	//Press Cancel
	IF	tyP0201OpsTravLifter.tyBarcodeScanner.tyBtnCancel.bRtCompl = TRUE THEN

		fUIInRtStatHide(ADR(tyP0201OpsTravLifter.tyBarcodeScanner.tyLyr.uiRtStat)); //hide
		IF tyP0201OpsTravLifter.tyQueryBoardInfo.tyBtnQueryBoardInfo.bValue THEN
		    fUIInRtStatOff(ADR(tyP0201OpsTravLifter.tyQueryBoardInfo.tyLyr.uiRtStat)); //show
		ELSIF tyP0201OpsTravLifter.tyCurrWorkOrderInfo.tyBtnQueryWorkOrderInfo.bValue THEN
			fUIInRtStatOff(ADR(tyP0201OpsTravLifter.tyQueryWorkOrderInfo.tyLyr.uiRtStat)); //show
		END_IF

		tyP0201OpsTravLifter.tyBarcodeScanner.tyStringBarcode.sValue :='';
		tyP0201OpsTravLifter.tyBarcodeScanner.tyStringTopBarcode.sValue :='';
		tyP0201OpsTravLifter.tyBarcodeScanner.tyStringTopBarcodeBK.sValue :='';
		tyP0201OpsTravLifter.tyBarcodeScanner.tyStringBottomBarcode.sValue :='';
		tyP0201OpsTravLifter.tyBarcodeScanner.tyStringBottomBarcodeBK.sValue :='';
		tyP0201OpsTravLifter.tyBarcodeScanner.tyStringMagazineBarcode.sValue :='';
		tyP0201OpsTravLifter.tyBarcodeScanner.tyStringMagazineBarcodeBK.sValue :='';
		tyP0201OpsTravLifter.tyBarcodeScanner.tyStringPCBBarcode.sValue :='';
		tyP0201OpsTravLifter.tyBarcodeScanner.tyStringPCBBarcodeBK.sValue :='';
		tyP0201OpsTravLifter.tyBarcodeScanner.tyBtnTop.bValue := FALSE;
		tyP0201OpsTravLifter.tyBarcodeScanner.tyBtnBottom.bValue := FALSE;
		tyP0201OpsTravLifter.tyBarcodeScanner.tyBtnMagazine.bValue := FALSE;
		tyP0201OpsTravLifter.tyBarcodeScanner.tyBtnPCB.bValue := FALSE;

		tyP0201OpsTravLifter.tyQueryBoardInfo.tyBtnBarcodeScanner.bValue := FALSE;
		tyP0201OpsTravLifter.tyQueryWorkOrderInfo.tyBtnBarcodeScanner.bValue := FALSE;

		tyP0201OpsTravLifter.tyBarcodeScanner.tyBtnCancel.bRtCompl := FALSE;
		tyP0201OpsTravLifter.tyBarcodeScanner.tyBtnCancel.bValue := FALSE;

	END_IF

END_ACTION
```

#### Act_OptP0201ChgParam.st
```iecst
ACTION Act_OptP0201ChgParam:
	//limit
	tyP0201OpsTravLifter.tyParam.tyNumMinSlt.diValueMax		:= tyP0201OpsTravLifter.tyParam.tyNumMaxSlt.diValue;
	tyP0201OpsTravLifter.tyParam.tyNumMaxSlt.diValueMin		:= tyP0201OpsTravLifter.tyParam.tyNumMinSlt.diValue;
	tyP0201OpsTravLifter.tyParam.tyNumPitch.diValueMax		:= tyP0201OpsTravLifter.tyParam.tyNumMaxSlt.diValue - tyP0201OpsTravLifter.tyParam.tyNumMinSlt.diValue + 1;
	tyP0201OpsTravLifter.tyParam.tyNumPitch.diValueMin		:= 1;

	tyP0201OpsTravLifter.tyParam.tyNumMinSltRear.diValueMax		:= tyP0201OpsTravLifter.tyParam.tyNumMaxSltRear.diValue;
	tyP0201OpsTravLifter.tyParam.tyNumMaxSltRear.diValueMin		:= tyP0201OpsTravLifter.tyParam.tyNumMinSltRear.diValue;
	tyP0201OpsTravLifter.tyParam.tyNumPitchRear.diValueMax		:= tyP0201OpsTravLifter.tyParam.tyNumMaxSltRear.diValue - tyP0201OpsTravLifter.tyParam.tyNumMinSltRear.diValue + 1;
	tyP0201OpsTravLifter.tyParam.tyNumPitchRear.diValueMin		:= 1;

	tyP0201OpsTravLifter.tyParam.tyNumMtrPshrExtSpd.diValueMin	:= p_tyNtParamCurr.tyProdRcpMtrPshrExtSpd.diMin;
	tyP0201OpsTravLifter.tyParam.tyNumMtrPshrExtSpd.diValueMax	:= p_tyNtParamCurr.tyProdRcpMtrPshrExtSpd.diMax;
	tyP0201OpsTravLifter.tyParam.tyNumMtrPshrExtTorq.diValueMin	:= p_tyNtParamCurr.tyProdRcpMtrPshrExtTorq.diMin;
	tyP0201OpsTravLifter.tyParam.tyNumMtrPshrExtTorq.diValueMax	:= p_tyNtParamCurr.tyProdRcpMtrPshrExtTorq.diMax;
	tyP0201OpsTravLifter.tyParam.tyNumPshrOffset.diValueMin		:= -(p_tyProdRcpCurrRcp2.diWidthInUM/2-p_tyMcParamCurr.diAWPusherAtHmPosInUM-5000 );
	tyP0201OpsTravLifter.tyParam.tyNumPshrOffset.diValueMax		:= (p_tyProdRcpCurrRcp2.diWidthInUM/2-p_tyMcParamCurr.diAWPusherAtHmPosInUM-5000 );

	//Control
	IF tyP0201OpsTravLifter.tyOps.tyBtnChgParam.bRtCompl = TRUE THEN
		tyP0201OpsTravLifter.tyOps.tyBtnChgParam.bRtCompl	:= FALSE;

		tyProdRcpCurrRcpWr	:= p_tyProdRcpCurrRcp0;

		tyP0201OpsTravLifter.tyParam.tyDrpDnMcMode.usiValueIdx	:= p_tyProdRcpCurrRcp0.usiMcMod;
		tyP0201OpsTravLifter.tyParam.tyNumMinSlt.diValue	:= p_tyProdRcpCurrRcp0.diMinSltValue;
		tyP0201OpsTravLifter.tyParam.tyNumMaxSlt.diValue	:= p_tyProdRcpCurrRcp0.diMaxSltValue;
		tyP0201OpsTravLifter.tyParam.tyNumPitch.diValue		:= p_tyProdRcpCurrRcp0.diPitch;

		tyP0201OpsTravLifter.tyParam.tyNumMinSltRear.diValue	:= p_tyProdRcpCurrRcp0.diMinSltValueRear;
		tyP0201OpsTravLifter.tyParam.tyNumMaxSltRear.diValue	:= p_tyProdRcpCurrRcp0.diMaxSltValueRear;
		tyP0201OpsTravLifter.tyParam.tyNumPitchRear.diValue		:= p_tyProdRcpCurrRcp0.diPitchRear;

		tyP0201OpsTravLifter.tyParam.tyNumMtrPshrExtSpd.diValue		:= p_tyProdRcpCurrRcp0.diMtrPshrExtSpd;
		tyP0201OpsTravLifter.tyParam.tyNumMtrPshrExtTorq.diValue	:= p_tyProdRcpCurrRcp0.diMtrPshrExtTorq;
		tyP0201OpsTravLifter.tyParam.tyNumPshrOffset.diValue		:= p_tyProdRcpCurrRcp0.diPshrOffset;

		fUIInRtStatOff(ADR(tyP0201OpsTravLifter.tyParam.tyLyr.uiRtStat));

	END_IF

	tyP0201OpsTravLifter.tyOps.tyBtnChgParam.bValue	:= tyP0201OpsTravLifter.tyParam.tyLyr.uiRtStat.0 = FALSE;

	IF tyP0201OpsTravLifter.tyParam.tyLyr.uiRtStat.0 = FALSE THEN

		IF tyP0201OpsTravLifter.tyParam.tyBtnSave.bRtCompl = TRUE THEN

			tyProdRcpCurrRcpWr.usiMcMod	:= tyP0201OpsTravLifter.tyParam.tyDrpDnMcMode.usiValueIdx;
			tyProdRcpCurrRcpWr.diMinSltValue := tyP0201OpsTravLifter.tyParam.tyNumMinSlt.diValue;
			tyProdRcpCurrRcpWr.diMaxSltValue := tyP0201OpsTravLifter.tyParam.tyNumMaxSlt.diValue;
			tyProdRcpCurrRcpWr.diPitch := tyP0201OpsTravLifter.tyParam.tyNumPitch.diValue;

			tyProdRcpCurrRcpWr.diMinSltValueRear := tyP0201OpsTravLifter.tyParam.tyNumMinSltRear.diValue;
			tyProdRcpCurrRcpWr.diMaxSltValueRear := tyP0201OpsTravLifter.tyParam.tyNumMaxSltRear.diValue;
			tyProdRcpCurrRcpWr.diPitchRear := tyP0201OpsTravLifter.tyParam.tyNumPitchRear.diValue;

			tyProdRcpCurrRcpWr.diMtrPshrExtSpd := tyP0201OpsTravLifter.tyParam.tyNumMtrPshrExtSpd.diValue;
			tyProdRcpCurrRcpWr.diMtrPshrExtTorq := tyP0201OpsTravLifter.tyParam.tyNumMtrPshrExtTorq.diValue;
			tyProdRcpCurrRcpWr.diPshrOffset := tyP0201OpsTravLifter.tyParam.tyNumPshrOffset.diValue;

			eProdRcpAct	:= ProdRcpActWriteCurrRcpParam;

			IF p_eProdRcpStatus = Done AND p_eProdRcpStat = ProdRcpActWriteCurrRcpParam THEN
				eProdRcpAct	:= ProdRcpActIdle;

				//UIP0400
				tyP0400ProdSel.tyProdSel.tyTxtMcMode.usiValueIdx	:= p_tyProdRcpCurrRcp0.usiMcMod;

				tyP0400ProdSel.tyProdSel.tyNumMinSlt.diValue	:= p_tyProdRcpCurrRcp0.diMinSltValue;
				tyP0400ProdSel.tyProdSel.tyNumMaxSlt.diValue	:= p_tyProdRcpCurrRcp0.diMaxSltValue;
				tyP0400ProdSel.tyProdSel.tyNumPitch.diValue		:= p_tyProdRcpCurrRcp0.diPitch;

				tyP0400ProdSel.tyProdSel.tyNumMinSltRear.diValue	:= p_tyProdRcpCurrRcp0.diMinSltValueRear;
				tyP0400ProdSel.tyProdSel.tyNumMaxSltRear.diValue	:= p_tyProdRcpCurrRcp0.diMaxSltValueRear;
				tyP0400ProdSel.tyProdSel.tyNumPitchRear.diValue		:= p_tyProdRcpCurrRcp0.diPitchRear;

				tyP0400ProdSel.tyProdSel.tyNumMtrPshrExtSpd.diValue		:= p_tyProdRcpCurrRcp0.diMtrPshrExtSpd;
				tyP0400ProdSel.tyProdSel.tyNumMtrPshrExtTorq.diValue	:= p_tyProdRcpCurrRcp0.diMtrPshrExtTorq;
				tyP0400ProdSel.tyProdSel.tyNumPshrOffset.diValue		:= p_tyProdRcpCurrRcp0.diPshrOffset;

				tyP0201OpsTravLifter.tyParam.tyBtnSave.bRtCompl	:= FALSE;
				tyP0201OpsTravLifter.tyParam.tyBtnSave.bValue	:= FALSE;

				fUIInRtStatHide(ADR(tyP0201OpsTravLifter.tyParam.tyLyr.uiRtStat));

			ELSIF p_eProdRcpStatus = Error THEN
				p_tyC0008MsgBox ACCESS ADR(tyP0201OpsTravLifter.tyMsgBoxSaveErr);

				IF tyP0201OpsTravLifter.tyMsgBoxSaveErr.tyBtnNo.bRtCompl = TRUE THEN
					tyP0201OpsTravLifter.tyMsgBoxSaveErr.tyBtnNo.bRtCompl	:= FALSE;
					tyP0201OpsTravLifter.tyMsgBoxSaveErr.tyBtnNo.bValue		:= FALSE;

					p_tyC0008MsgBox ACCESS ADR(tyP0201OpsTravLifter.tyMsgBoxHide);

					//Restore Param
					tyProdRcpCurrRcpWr	:= p_tyProdRcpCurrRcp0;

					tyP0201OpsTravLifter.tyParam.tyBtnSave.bRtCompl	:= FALSE;
					tyP0201OpsTravLifter.tyParam.tyBtnSave.bValue	:= FALSE;

					fUIInRtStatHide(ADR(tyP0201OpsTravLifter.tyParam.tyLyr.uiRtStat));

				END_IF

			END_IF

		ELSIF tyP0201OpsTravLifter.tyParam.tyBtnCancel.bRtCompl = TRUE THEN
			tyP0201OpsTravLifter.tyParam.tyBtnCancel.bRtCompl	:= FALSE;
			tyP0201OpsTravLifter.tyParam.tyBtnCancel.bValue		:= FALSE;

			fUIInRtStatHide(ADR(tyP0201OpsTravLifter.tyParam.tyLyr.uiRtStat));

		END_IF

	END_IF

	//Mask
	tyP0201OpsTravLifter.tyOps.tyBtnChgParam.uiMaskRtStat.0	:= p_tyUsrMgmtCurrAccessRgt.bChgParam AND p_bOpsStatusStop;

END_ACTION
```

#### Act_OptP0201CurrWorkOrderInfo.st
```iecst
ACTION Act_OptP0201CurrWorkOrderInfo:

	//Hide or Unhide UI button
	IF p_tyHermesConfiguration.tySvyParam.bFeatureQueryWorkOrderInfo = TRUE AND p_tyNtParamCurr.bHermesSvyPrep AND p_tyMcParamCurr.bHermesSvyEn AND p_tyNtParamCurr.bHermesSvyFirstMcInTheLine AND
		p_tyNtParamCurr.bProjAutoRcpPrep = FALSE THEN
		fUIInRtStatOff(ADR(tyP0201OpsTravLifter.tyCurrWorkOrderInfo.tyBtnQueryWorkOrderInfo.uiRtStat)); //show
	ELSE
		fUIInRtStatHide(ADR(tyP0201OpsTravLifter.tyCurrWorkOrderInfo.tyBtnQueryWorkOrderInfo.uiRtStat)); //hide
		tyP0201OpsTravLifter.tyCurrWorkOrderInfo.tyBtnQueryWorkOrderInfo.bValue := FALSE;
	END_IF

	//Press Query Work Order Info button, bValue will toggle.
	IF tyP0201OpsTravLifter.tyCurrWorkOrderInfo.tyBtnQueryWorkOrderInfo.bRtCompl = TRUE THEN
		tyP0201OpsTravLifter.tyCurrWorkOrderInfo.tyBtnQueryWorkOrderInfo.bRtCompl := FALSE;
	END_IF

	//Popup
	IF 	EDGEPOS (tyP0201OpsTravLifter.tyCurrWorkOrderInfo.tyBtnQueryWorkOrderInfo.bValue = TRUE) THEN
		fUIInRtStatOff(ADR(tyP0201OpsTravLifter.tyCurrWorkOrderInfo.tyLyr.uiRtStat)); //show popup View WorkOrder
		fUIInRtStatHide(ADR(tyP0201OpsTravLifter.tyBarcodeScanner.tyLyr.uiRtStat)); //hide popup BCScanner
		fUIInRtStatHide(ADR(tyP0201OpsTravLifter.tyQueryWorkOrderInfo.tyLyr.uiRtStat)); //hide popup QueryWorkOrder
	END_IF

	//Reset
	IF tyP0201OpsTravLifter.tyCurrWorkOrderInfo.tyBtnQueryWorkOrderInfo.bValue = FALSE THEN
		bQueryWorkOrderInfo := FALSE;
	END_IF

	//Press Query button, go page QueryWorkOrderInfo
	IF	tyP0201OpsTravLifter.tyCurrWorkOrderInfo.tyBtnQuery.bRtCompl = TRUE AND p_tyNtParamCurr.eCustomerReq = Siemens (*AND bDummy *)THEN

		fUIInRtStatHide(ADR(tyP0201OpsTravLifter.tyCurrWorkOrderInfo.tyLyr.uiRtStat)); //hide popup View WorkOrder
		fUIInRtStatHide(ADR(tyP0201OpsTravLifter.tyBarcodeScanner.tyLyr.uiRtStat)); //hide popup BCScanner
		fUIInRtStatOff(ADR(tyP0201OpsTravLifter.tyQueryWorkOrderInfo.tyLyr.uiRtStat)); //show popup QueryWorkOrder

//		bQueryWorkOrderInfo := TRUE;                                                                  //ADD
//		tyP0201OpsTravLifter.tyCurrWorkOrderInfo.tyBtnQueryWorkOrderInfo.bValue := TRUE;

		tyP0201OpsTravLifter.tyCurrWorkOrderInfo.tyBtnQuery.bValue   := FALSE;
		tyP0201OpsTravLifter.tyCurrWorkOrderInfo.tyBtnQuery.bRtCompl := FALSE;

//	ELSE                                                                                            //ADD
//		bQueryWorkOrderInfo := FALSE;
//		tyP0201OpsTravLifter.tyCurrWorkOrderInfo.tyBtnQueryWorkOrderInfo.bValue := FALSE;
	ELSIF tyP0201OpsTravLifter.tyCurrWorkOrderInfo.tyBtnQuery.bRtCompl = TRUE AND p_tyNtParamCurr.eCustomerReq = Siemens THEN	        //ADD 2022-0780A
		fUIInRtStatHide(ADR(tyP0201OpsTravLifter.tyCurrWorkOrderInfo.tyLyr.uiRtStat)); //hide popup View WorkOrder
		bQueryWorkOrderInfo := TRUE;

		tyP0201OpsTravLifter.tyCurrWorkOrderInfo.tyBtnQuery.bValue   := FALSE;
		tyP0201OpsTravLifter.tyCurrWorkOrderInfo.tyBtnQuery.bRtCompl := FALSE;
	END_IF

//	IF p_tyNtParamCurr.eCustomerReq = Siemens AND p_bAllZonesEmpty AND p_bOpsConvWaitForTopUpBrd AND  bBypassCoverSwitch = FALSE AND  bTopUpBrdRdy = FALSE AND p_sWorkOrderId <>''  THEN
//		fUIInRtStatHide(ADR(tyP0201OpsTravLifter.tyCurrWorkOrderInfo.tyBtnQuery.uiRtStat)); //hide
//		fUIInRtStatOff(ADR(tyP0201OpsTravLifter.tyCurrWorkOrderInfo.tyBtnDelete.uiRtStat)); //Show
//	ELSIF (*p_bSiemensMcModeChgPrep AND*) p_bAllZonesEmpty AND p_bOpsConvWaitForTopUpBrd AND bBypassCoverSwitch = FALSE AND  bTopUpBrdRdy = FALSE AND p_sWorkOrderId = '' THEN
//		fUIInRtStatOff(ADR(tyP0201OpsTravLifter.tyCurrWorkOrderInfo.tyBtnQuery.uiRtStat)); //Show
//		fUIInRtStatHide(ADR(tyP0201OpsTravLifter.tyCurrWorkOrderInfo.tyBtnDelete.uiRtStat)); //Hide
//	ELSE
//		fUIInRtStatHide(ADR(tyP0201OpsTravLifter.tyCurrWorkOrderInfo.tyBtnQuery.uiRtStat)); //Show
//		fUIInRtStatHide(ADR(tyP0201OpsTravLifter.tyCurrWorkOrderInfo.tyBtnDelete.uiRtStat)); //Hide
//	END_IF

	//Press Exit
	IF	tyP0201OpsTravLifter.tyCurrWorkOrderInfo.tyBtnExit.bRtCompl = TRUE THEN

		fUIInRtStatHide(ADR(tyP0201OpsTravLifter.tyCurrWorkOrderInfo.tyLyr.uiRtStat)); //hide popup View WorkOrder
		fUIInRtStatHide(ADR(tyP0201OpsTravLifter.tyBarcodeScanner.tyLyr.uiRtStat)); //hide popup BCScanner
		fUIInRtStatHide(ADR(tyP0201OpsTravLifter.tyQueryWorkOrderInfo.tyLyr.uiRtStat)); //hide popup QueryWorkOrder

		tyP0201OpsTravLifter.tyCurrWorkOrderInfo.tyBtnQueryWorkOrderInfo.bValue := FALSE;

		tyP0201OpsTravLifter.tyCurrWorkOrderInfo.tyBtnExit.bValue   := FALSE;
		tyP0201OpsTravLifter.tyCurrWorkOrderInfo.tyBtnExit.bRtCompl := FALSE;
	END_IF

	tyP0201OpsTravLifter.tyCurrWorkOrderInfo.tyStringWorkOrder.sValue := p_sWorkOrderId;

	//Press Delete, prompt confirm to delete
	IF	tyP0201OpsTravLifter.tyCurrWorkOrderInfo.tyBtnDelete.bRtCompl = TRUE THEN
		p_tyC0008MsgBox ACCESS ADR(tyP0201OpsTravLifter.tyMsgBoxAskDelete);

		IF tyP0201OpsTravLifter.tyMsgBoxAskDelete.tyBtnYes.bRtCompl THEN
		   tyP0201OpsTravLifter.tyMsgBoxAskDelete.tyBtnYes.bRtCompl := FALSE;
			bDeleteWorkOrder := TRUE;
			tyP0201OpsTravLifter.tyCurrWorkOrderInfo.tyBtnDelete.bValue := FALSE;
			tyP0201OpsTravLifter.tyCurrWorkOrderInfo.tyBtnDelete.bRtCompl := FALSE;
			p_tyC0008MsgBox ACCESS ADR(tyP0201OpsTravLifter.tyMsgBoxHide);
			tyP0201OpsTravLifter.tyMsgBoxAskDelete.tyBtnYes.bValue := FALSE;

		ELSIF tyP0201OpsTravLifter.tyMsgBoxAskDelete.tyBtnNo.bRtCompl THEN
			tyP0201OpsTravLifter.tyMsgBoxAskDelete.tyBtnNo.bRtCompl := FALSE;

			bDeleteWorkOrder := FALSE;
			tyP0201OpsTravLifter.tyCurrWorkOrderInfo.tyBtnDelete.bValue := FALSE;
			tyP0201OpsTravLifter.tyCurrWorkOrderInfo.tyBtnDelete.bRtCompl := FALSE;
			p_tyC0008MsgBox ACCESS ADR(tyP0201OpsTravLifter.tyMsgBoxHide);
			tyP0201OpsTravLifter.tyMsgBoxAskDelete.tyBtnNo.bValue := FALSE;
		END_IF

	END_IF

	//Bitmap
	IF tyP0201OpsTravLifter.tyCurrWorkOrderInfo.tyBtnQueryWorkOrderInfo.bValue THEN
		tyP0201OpsTravLifter.tyCurrWorkOrderInfo.tyBtnQueryWorkOrderInfo.usiBitmapIdx := 1;
	ELSE
		tyP0201OpsTravLifter.tyCurrWorkOrderInfo.tyBtnQueryWorkOrderInfo.usiBitmapIdx := 0;
	END_IF

END_ACTION
```

#### Act_OptP0201IOMonitor.st
```iecst
ACTION Act_OptP0201IOMonitor:

	IF tyP0201OpsTravLifter.tyOps.tyHotspotIOMonitor.bRtCompl = TRUE THEN
		tyP0201OpsTravLifter.tyOps.tyHotspotIOMonitor.bRtCompl	:= FALSE;

		fUIInRtStatOff(ADR(tyP0201OpsTravLifter.tyIOMonitor.tyLyr.uiRtStat));
		fUIInRtStatHide(ADR(tyP0201OpsTravLifter.tyOps.tyLyrProdRear.uiRtStat));

		p_tyC0004Navi ACCESS ADR(tyP0201OpsTravLifter.tyNaviHide);

	ELSIF tyP0201OpsTravLifter.tyIOMonitor.tyHotspotClose.bRtCompl = TRUE THEN
		tyP0201OpsTravLifter.tyIOMonitor.tyHotspotClose.bRtCompl	:= FALSE;

		fUIInRtStatHide(ADR(tyP0201OpsTravLifter.tyIOMonitor.tyLyr.uiRtStat));
		IF p_tyNtParamCurr.eProjMag = LDMagQuadruple THEN
			fUIInRtStatOff(ADR(tyP0201OpsTravLifter.tyOps.tyLyrProdRear.uiRtStat));
		ELSE
			fUIInRtStatHide(ADR(tyP0201OpsTravLifter.tyOps.tyLyrProdRear.uiRtStat));
		END_IF
		p_tyC0004Navi ACCESS ADR(tyP0201OpsTravLifter.tyNaviBack);

	END_IF

	IF tyP0201OpsTravLifter.tyIOMonitor.tyLyr.uiRtStat.0 = FALSE THEN

		//Digital Input
		tyP0201OpsTravLifter.tyIOMonitor.tyBtnSafetyRlySig.bValue			:= p_tyDI.bSafetyRlySig;
		tyP0201OpsTravLifter.tyIOMonitor.tyBtnEStop.bValue					:= p_tyDI.bEStopSig;
		tyP0201OpsTravLifter.tyIOMonitor.tyBtnCoverSWSig.bValue				:= p_tyDI.bCoverSWSig;
		tyP0201OpsTravLifter.tyIOMonitor.tyBtnDSBA.bValue					:= p_tyDI.bDSBA;
		tyP0201OpsTravLifter.tyIOMonitor.tyBtnDSBB.bValue					:= p_tyDI.bDSBB;
		tyP0201OpsTravLifter.tyIOMonitor.tyBtnPullerExtRS.bValue			:= p_tyDI.bPullerExtRS;
		tyP0201OpsTravLifter.tyIOMonitor.tyBtnPullerRetRS.bValue			:= p_tyDI.bPullerRetRS;
		tyP0201OpsTravLifter.tyIOMonitor.tyBtnPullerRotCylHmRS.bValue		:= p_tyDI.bPullerRotHmRS;
		tyP0201OpsTravLifter.tyIOMonitor.tyBtnPullerRotCylRmRS.bValue		:= p_tyDI.bPullerRotRmRS;
		tyP0201OpsTravLifter.tyIOMonitor.tyBtnConvLftSen.bValue				:= p_tyDI.bConvLftSen;
		tyP0201OpsTravLifter.tyIOMonitor.tyBtnConvRgtSen.bValue				:= p_tyDI.bConvRgtSen;
		tyP0201OpsTravLifter.tyIOMonitor.tyBtnLifterTmBeltSen.bValue		:= p_tyDI.bLifterTimingBeltSen;
		tyP0201OpsTravLifter.tyIOMonitor.tyBtnLifterSafetyLmtSw1.bValue		:= p_tyDI.bLifterSafetyLmtSW1;
		tyP0201OpsTravLifter.tyIOMonitor.tyBtnLifterSafetyLmtSw2.bValue		:= p_tyDI.bLifterSafetyLmtSW2;
		tyP0201OpsTravLifter.tyIOMonitor.tyBtnInletShutterOpenSen.bValue	:= p_tyDI.bInShutterOpenRS;
		tyP0201OpsTravLifter.tyIOMonitor.tyBtnInletShutterCloseSen.bValue	:= p_tyDI.bInShutterCloseRS;
		tyP0201OpsTravLifter.tyIOMonitor.tyBtnOutletShutterOpenSen.bValue	:= p_tyDI.bOutShutterOpenRS;
		tyP0201OpsTravLifter.tyIOMonitor.tyBtnOutletShutterCloseSen.bValue	:= p_tyDI.bOutShutterCloseRS;
		tyP0201OpsTravLifter.tyIOMonitor.tyBtnAntiJamSen.bValue				:= p_tyDI.bPullerAntiJam;

		tyP0201OpsTravLifter.tyIOMonitor.tyBtnInletShutterCloseSen2.bValue	:= p_tyDI.bInShutterCloseRS2;
		tyP0201OpsTravLifter.tyIOMonitor.tyBtnInletShutterCloseSen3.bValue	:= p_tyDI.bInShutterCloseRS3;
		tyP0201OpsTravLifter.tyIOMonitor.tyBtnInletShutterOpenSen2.bValue	:= p_tyDI.bInShutterOpenRS2;
		tyP0201OpsTravLifter.tyIOMonitor.tyBtnInletShutterOpenSen3.bValue	:= p_tyDI.bInShutterOpenRS3;
		tyP0201OpsTravLifter.tyIOMonitor.tyBtnOutletShutterOpenSen2.bValue	:= p_tyDI.bOutShutterCloseRS2;
		tyP0201OpsTravLifter.tyIOMonitor.tyBtnOutletShutterOpenSen2.bValue	:= p_tyDI.bOutShutterOpenRS2;

		tyP0201OpsTravLifter.tyIOMonitor.tyBtnBypCurtainSensorPB.bValue		:= p_tyDI.bBypCurtainSensorPB;
		tyP0201OpsTravLifter.tyIOMonitor.tyBtnConvClrSen.bValue				:= p_tyDI.bConvClrSen;
		tyP0201OpsTravLifter.tyIOMonitor.tyBtnMagWidthChk.bValue			:= p_tyDI.bMagWidthChkSen;
		tyP0201OpsTravLifter.tyIOMonitor.tyBtnSafetySigDS.bValue			:= p_tyDI.bDSSafetySig;
		tyP0201OpsTravLifter.tyIOMonitor.tyBtnUnlockSigDS.bValue			:= p_tyDI.bDSUnlockCoverSig;

		//Digital Output
		tyP0201OpsTravLifter.tyIOMonitor.tyBtnSafetyRlyRst.bValue			:= p_tyDO.bSafetyRlyRst;
		tyP0201OpsTravLifter.tyIOMonitor.tyBtnTLGreen.bValue				:= p_tyDO.bTLGreen;
		tyP0201OpsTravLifter.tyIOMonitor.tyBtnTLAmber.bValue				:= p_tyDO.bTLAmber;
		tyP0201OpsTravLifter.tyIOMonitor.tyBtnTLRed.bValue					:= p_tyDO.bTLRed;
		tyP0201OpsTravLifter.tyIOMonitor.tyBtnBuzzer.bValue					:= p_tyDO.bBuzzer;
		tyP0201OpsTravLifter.tyIOMonitor.tyBtnDBAA.bValue					:= p_tyDO.bDBAA;
		tyP0201OpsTravLifter.tyIOMonitor.tyBtnDBAB.bValue					:= p_tyDO.bDBAB;
		tyP0201OpsTravLifter.tyIOMonitor.tyBtnPullerExtCtrl.bValue			:= p_tyDO.bPullerExtCtrl;
		tyP0201OpsTravLifter.tyIOMonitor.tyBtnPullerRetCtrl.bValue			:= p_tyDO.bPullerRetCtrl;
		tyP0201OpsTravLifter.tyIOMonitor.tyBtnRotPullerCtrl.bValue			:= p_tyDO.bRotPullerCtrl;
		tyP0201OpsTravLifter.tyIOMonitor.tyBtnInShutterOpenCtrl.bValue		:= p_tyDO.bInShutterOpenCtrl;
		tyP0201OpsTravLifter.tyIOMonitor.tyBtnInShutterCloseCtrl.bValue		:= p_tyDO.bInShutterCloseCtrl;
		tyP0201OpsTravLifter.tyIOMonitor.tyBtnOutShutterOpenCtrl.bValue		:= p_tyDO.bOutShutterOpenCtrl;
		tyP0201OpsTravLifter.tyIOMonitor.tyBtnOutShutterCloseCtrl.bValue	:= p_tyDO.bOutShutterCloseCtrl;
		tyP0201OpsTravLifter.tyIOMonitor.tyBtnPullerConvMtrOn.bValue		:= p_tyDO.bPullConvMtrOn;

		tyP0201OpsTravLifter.tyIOMonitor.tyBtnInShutterCloseCtrl2.bValue	:= p_tyDO.bInShutterCloseCtrl2;
		tyP0201OpsTravLifter.tyIOMonitor.tyBtnInShutterOpenCtrl2.bValue		:= p_tyDO.bInShutterOpenCtrl2;
		tyP0201OpsTravLifter.tyIOMonitor.tyBtnInShutterCloseCtrl3.bValue	:= p_tyDO.bInShutterCloseCtrl3;
		tyP0201OpsTravLifter.tyIOMonitor.tyBtnInShutterOpenCtrl3.bValue		:= p_tyDO.bInShutterOpenCtrl3;
		tyP0201OpsTravLifter.tyIOMonitor.tyBtnOutShutterCloseCtrl2.bValue	:= p_tyDO.bOutShutterCloseCtrl2;
		tyP0201OpsTravLifter.tyIOMonitor.tyBtnOutShutterOpenCtrl2.bValue	:= p_tyDO.bOutShutterOpenCtrl2;

		tyP0201OpsTravLifter.tyIOMonitor.tyBtnBypCurtainSensorCtrl.bValue	:= p_tyDO.bBypCurtainSen;
		tyP0201OpsTravLifter.tyIOMonitor.tyBtnRstCurtainSensor.bValue		:= p_tyDO.bRstCurtainSen;
		tyP0201OpsTravLifter.tyIOMonitor.tyBtnSftySglToUSDS.bValue			:= p_tyDO.bMcSafetySigToDS;

	END_IF

END_ACTION
```

#### Act_OptP0201QueryBoardInfo.st
```iecst
ACTION Act_OptP0201QueryBoardInfo:

	//Hide or Unhide UI button
//	IF p_tyHermesConfiguration.a_tyUSParam[0].bFeatureQueryBoardInfo = TRUE AND p_tyNtParamCurr.bHermesPrep AND p_tyMcParamCurr.eUSComm = McSetCommModHermes THEN
//		fUIInRtStatOff(ADR(tyP0201OpsTravLifter.tyQueryBoardInfo.tyBtnQueryBoardInfo.uiRtStat)); //show
//	ELSE
		fUIInRtStatHide(ADR(tyP0201OpsTravLifter.tyQueryBoardInfo.tyBtnQueryBoardInfo.uiRtStat)); //hide
//		tyP0201OpsTravLifter.tyQueryBoardInfo.tyBtnQueryBoardInfo.bValue := FALSE;
//	END_IF

	//Mask
	IF p_tyNtParamCurr.bHermesScannerPrep = TRUE AND p_tyMcParamCurr.bHermesScannerEn = TRUE THEN
		fUIInRtStatHide(ADR(tyP0201OpsTravLifter.tyQueryBoardInfo.tyBtnBarcodeScanner.uiMaskRtStat)); //hide the mask
	ELSE
		fUIInRtStatOff(ADR(tyP0201OpsTravLifter.tyQueryBoardInfo.tyBtnBarcodeScanner.uiMaskRtStat)); //show the mask
	END_IF

	//Press Query Board Info button, bValue will toggle 0,1,0,1.
	IF tyP0201OpsTravLifter.tyQueryBoardInfo.tyBtnQueryBoardInfo.bRtCompl = TRUE THEN
		tyP0201OpsTravLifter.tyQueryBoardInfo.tyBtnQueryBoardInfo.bRtCompl := FALSE;
	END_IF

	//Popup
	IF 	EDGEPOS (tyP0201OpsTravLifter.tyQueryBoardInfo.tyBtnQueryBoardInfo.bValue = TRUE) THEN
		fUIInRtStatOff(ADR(tyP0201OpsTravLifter.tyQueryBoardInfo.tyLyr.uiRtStat)); //show popup QueryBoardInfo
		fUIInRtStatHide(ADR(tyP0201OpsTravLifter.tyBarcodeScanner.tyLyr.uiRtStat)); //hide popup BCScanner
	END_IF

	IF 	EDGEPOS (tyP0201OpsTravLifter.tyQueryBoardInfo.tyBtnBarcodeScanner.bValue = TRUE) THEN
		fUIInRtStatHide(ADR(tyP0201OpsTravLifter.tyQueryBoardInfo.tyLyr.uiRtStat)); //hide popup QueryBoardInfo
		fUIInRtStatOff(ADR(tyP0201OpsTravLifter.tyBarcodeScanner.tyLyr.uiRtStat)); //show popup BCScanner
		fUIInRtStatHide(ADR(tyP0201OpsTravLifter.tyBarcodeScanner.tyBtnTop.uiMaskRtStat)); //hide Mask Top
		fUIInRtStatOff(ADR(tyP0201OpsTravLifter.tyBarcodeScanner.tyBtnMagazine.uiMaskRtStat)); //Mask Magazine
	END_IF

	//Press OK, set bQueryBoardInfo

	IF	tyP0201OpsTravLifter.tyQueryBoardInfo.tyBtnOk.bRtCompl = TRUE THEN

		fUIInRtStatHide(ADR(tyP0201OpsTravLifter.tyQueryBoardInfo.tyLyr.uiRtStat)); //close popup

	    IF (tyP0201OpsTravLifter.tyQueryBoardInfo.tyStringTopBarcode.sValue <> '') OR (tyP0201OpsTravLifter.tyQueryBoardInfo.tyStringBottomBarcode.sValue <> '') THEN

			bQueryBoardInfo := TRUE;
			tyP0201OpsTravLifter.tyQueryBoardInfo.tyBtnQueryBoardInfo.bValue := TRUE;
		ELSE
			bQueryBoardInfo := FALSE;
			tyP0201OpsTravLifter.tyQueryBoardInfo.tyBtnQueryBoardInfo.bValue := FALSE;
		END_IF

		tyP0201OpsTravLifter.tyQueryBoardInfo.tyBtnOk.bValue := FALSE;

		tyP0201OpsTravLifter.tyQueryBoardInfo.tyBtnOk.bRtCompl := FALSE;

	END_IF

	//Reset
	IF tyP0201OpsTravLifter.tyQueryBoardInfo.tyBtnQueryBoardInfo.bValue = FALSE THEN
		bQueryBoardInfo := FALSE;
	END_IF

    //Press Cancel
	IF	tyP0201OpsTravLifter.tyQueryBoardInfo.tyBtnCancel.bRtCompl = TRUE THEN

		fUIInRtStatHide(ADR(tyP0201OpsTravLifter.tyQueryBoardInfo.tyLyr.uiRtStat)); //hide

		tyP0201OpsTravLifter.tyQueryBoardInfo.tyBtnQueryBoardInfo.bValue := FALSE;

		tyP0201OpsTravLifter.tyQueryBoardInfo.tyBtnCancel.bRtCompl := FALSE;
		tyP0201OpsTravLifter.tyQueryBoardInfo.tyBtnCancel.bValue := FALSE;
	END_IF

	//Bitmap
	IF tyP0201OpsTravLifter.tyQueryBoardInfo.tyBtnQueryBoardInfo.bValue THEN
		tyP0201OpsTravLifter.tyQueryBoardInfo.tyBtnQueryBoardInfo.usiBitmapIdx := 1;
	ELSE
		tyP0201OpsTravLifter.tyQueryBoardInfo.tyBtnQueryBoardInfo.usiBitmapIdx := 0;
	END_IF

END_ACTION
```
